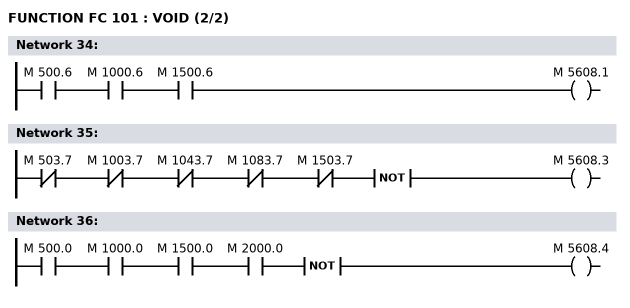

      A     M    500.6;
      A     M   1000.6;
      A     M   1500.6;
      =     M   5608.1;
NETWORK
TITLE =

      AN    M    503.7;
      AN    M   1003.7;
      AN    M   1043.7;
      AN    M   1083.7;
      AN    M   1503.7;
      NOT   ;
      =     M   5608.3;
NETWORK
TITLE =

      A     M    500.0;
      A     M   1000.0;
      A     M   1500.0;
      A     M   2000.0;
      NOT   ;
      =     M   5608.4;
NETWORK
TITLE =

      AN    OV;
      =     L      0.0;
      A     L      0.0;
      JNB   _001;
      L     ID  1302;
      T     MD  5610;
_001: NOP   0;
      A     L      0.0;
      JNB   _002;
      L     ID  1306;
      T     MD  5614;
_002: NOP   0;
      A     L      0.0;
      JNB   _003;
      L     ID  1310;
      T     MW  5618;
_003: NOP   0;
NETWORK
TITLE =

      AN    OV;
      =     L      0.0;
      A     L      0.0;
      A     I   1301.4;
      L     S5T#2S;
      SD    T     90;
      A     L      0.0;
      AN    I   1301.4;
      L     S5T#2S;
      SD    T     91;
NETWORK
TITLE =
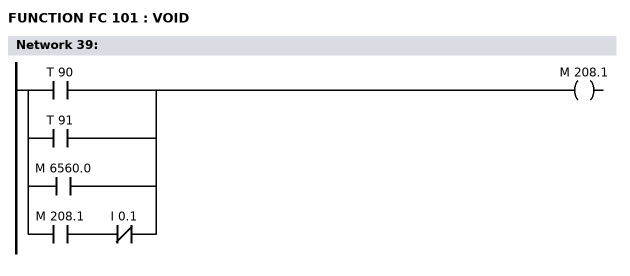

      O     T     90;
      O     T     91;
      O     M   6560.0;
      O     ;
      A     M    208.1;
      AN    I      0.1;
      =     M    208.1;
END_FUNCTION

FUNCTION_BLOCK FB 108
TITLE =
VERSION : 0.1

BEGIN
NETWORK
TITLE =PROFINET ERROR(1~10)
//
//
      A     M      3.3;
      =     L      0.0;
      A     L      0.0;
      A(    ;
      O     DB327.DBX 1025.3;
      O     ;
      A     M   7000.0;
      AN    I      0.1;
      AN    I    113.3;
      AN    I    317.3;
      AN    I    205.3;
      )     ;
      =     L      0.1;
      A     L      0.1;
      A     T    700;
      =     M   7000.0;
      A     L      0.1;
      BLD   102;
      L     S5T#0MS;
      SD    T    700;
      A     L      0.0;
      A(    ;
      O     DB327.DBX 1027.3;
      O     ;
      A     M   7000.1;
      AN    I      0.1;
      AN    I    113.3;
      AN    I    317.3;
      AN    I    205.3;
      )     ;
      =     L      0.1;
      A     L      0.1;
      A     T    701;
      =     M   7000.1;
      A     L      0.1;
      BLD   102;
      L     S5T#0MS;
      SD    T    701;
      A     L      0.0;
      A(    ;
      O     DB327.DBX 1029.3;
      O     ;
      A     M   7000.2;
      AN    I      0.1;
      AN    I    113.3;
      AN    I    317.3;
      AN    I    205.3;
      )     ;
      =     L      0.1;
      A     L      0.1;
      A     T    702;
      =     M   7000.2;
      A     L      0.1;
      BLD   102;
      L     S5T#0MS;
      SD    T    702;
      A     L      0.0;
      A(    ;
      O     DB327.DBX 1031.3;
      O     ;
      A     M   7000.3;
      AN    I      0.1;
      AN    I    113.3;
      AN    I    317.3;
      AN    I    205.3;
      )     ;
      =     L      0.1;
      A     L      0.1;
      A     T    703;
      =     M   7000.3;
      A     L      0.1;
      BLD   102;
      L     S5T#0MS;
      SD    T    703;
      A     L      0.0;
      A(    ;
      O     DB327.DBX 1033.3;
      O     ;
      A     M   7000.4;
      AN    I      0.1;
      AN    I    113.3;
      AN    I    317.3;
      AN    I    205.3;
      )     ;
      =     L      0.1;
      A     L      0.1;
      A     T    704;
      =     M   7000.4;
      A     L      0.1;
      BLD   102;
      L     S5T#0MS;
      SD    T    704;
      A     L      0.0;
      A(    ;
      O     DB327.DBX 1035.3;
      O     ;
      A     M   7000.5;
      AN    I      0.1;
      AN    I    113.3;
      AN    I    317.3;
      AN    I    205.3;
      )     ;
      =     L      0.1;
      A     L      0.1;
      A     T    705;
      =     M   7000.5;
      A     L      0.1;
      BLD   102;
      L     S5T#0MS;
      SD    T    705;
      A     L      0.0;
      A(    ;
      O     DB327.DBX 1037.3;
      O     ;
      A     M   7000.6;
      AN    I      0.1;
      AN    I    113.3;
      AN    I    317.3;
      AN    I    205.3;
      )     ;
      =     L      0.1;
      A     L      0.1;
      A     T    706;
      =     M   7000.6;
      A     L      0.1;
      BLD   102;
      L     S5T#0MS;
      SD    T    706;
      A     L      0.0;
      A(    ;
      O     DB327.DBX 1039.3;
      O     ;
      A     M   7000.7;
      AN    I      0.1;
      AN    I    113.3;
      AN    I    317.3;
      AN    I    205.3;
      )     ;
      =     L      0.1;
      A     L      0.1;
      A     T    707;
      =     M   7000.7;
      A     L      0.1;
      BLD   102;
      L     S5T#0MS;
      SD    T    707;
      A     L      0.0;
      A(    ;
      O     DB327.DBX 1041.3;
      O     ;
      A     M   7001.0;
      AN    I      0.1;
      AN    I    113.3;
      AN    I    317.3;
      AN    I    205.3;
      )     ;
      =     L      0.1;
      A     L      0.1;
      A     T    708;
      =     M   7001.0;
      A     L      0.1;
      BLD   102;
      L     S5T#0MS;
      SD    T    708;
      A     L      0.0;
      A(    ;
      O     DB327.DBX 1043.3;
      O     ;
      A     M   7001.1;
      AN    I      0.1;
      AN    I    113.3;
      AN    I    317.3;
      AN    I    205.3;
      )     ;
      =     L      0.1;
      A     L      0.1;
      A     T    709;
      =     M   7001.1;
      A     L      0.1;
      BLD   102;
      L     S5T#0MS;
      SD    T    709;
NETWORK
TITLE =PROFINET ERROR(11~20)
//
//
      A     M      3.3;
      =     L      0.0;
      A     L      0.0;
      A(    ;
      O     DB327.DBX 1045.3;
      O     ;
      A     M   7001.2;
      AN    I      0.1;
      AN    I    113.3;
      AN    I    317.3;
      AN    I    205.3;
      )     ;
      =     L      0.1;
      A     L      0.1;
      A     T    710;
      =     M   7001.2;
      A     L      0.1;
      BLD   102;
      L     S5T#0MS;
      SD    T    710;
      A     L      0.0;
      A(    ;
      O     DB327.DBX 1047.3;
      O     ;
      A     M   7001.3;
      AN    I      0.1;
      AN    I    113.3;
      AN    I    317.3;
      AN    I    205.3;
      )     ;
      =     L      0.1;
      A     L      0.1;
      A     T    711;
      =     M   7001.3;
      A     L      0.1;
      BLD   102;
      L     S5T#0MS;
      SD    T    711;
      A     L      0.0;
      A(    ;
      O     DB327.DBX 1049.3;
      O     ;
      A     M   7001.4;
      AN    I      0.1;
      AN    I    113.3;
      AN    I    317.3;
      AN    I    205.3;
      )     ;
      =     L      0.1;
      A     L      0.1;
      A     T    712;
      =     M   7001.4;
      A     L      0.1;
      BLD   102;
      L     S5T#0MS;
      SD    T    712;
      A     L      0.0;
      A(    ;
      O     DB327.DBX 1051.3;
      O     ;
      A     M   7001.5;
      AN    I      0.1;
      AN    I    113.3;
      AN    I    317.3;
      AN    I    205.3;
      )     ;
      =     L      0.1;
      A     L      0.1;
      A     T    713;
      =     M   7001.5;
      A     L      0.1;
      BLD   102;
      L     S5T#0MS;
      SD    T    713;
      A     L      0.0;
      A(    ;
      O     DB327.DBX 1053.3;
      O     ;
      A     M   7001.6;
      AN    I      0.1;
      AN    I    113.3;
      AN    I    317.3;
      AN    I    205.3;
      )     ;
      =     L      0.1;
      A     L      0.1;
      A     T    714;
      =     M   7001.6;
      A     L      0.1;
      BLD   102;
      L     S5T#0MS;
      SD    T    714;
      A     L      0.0;
      A(    ;
      O     DB327.DBX 1055.3;
      O     ;
      A     M   7001.7;
      AN    I      0.1;
      AN    I    113.3;
      AN    I    317.3;
      AN    I    205.3;
      )     ;
      =     L      0.1;
      A     L      0.1;
      A     T    715;
      =     M   7001.7;
      A     L      0.1;
      BLD   102;
      L     S5T#0MS;
      SD    T    715;
      A     L      0.0;
      A(    ;
      O     DB327.DBX 1057.3;
      O     ;
      A     M   7002.0;
      AN    I      0.1;
      AN    I    113.3;
      AN    I    317.3;
      AN    I    205.3;
      )     ;
      =     L      0.1;
      A     L      0.1;
      A     T    716;
      =     M   7002.0;
      A     L      0.1;
      BLD   102;
      L     S5T#0MS;
      SD    T    716;
      A     L      0.0;
      A(    ;
      O     DB327.DBX 1059.3;
      O     ;
      A     M   7002.1;
      AN    I      0.1;
      AN    I    113.3;
      AN    I    317.3;
      AN    I    205.3;
      )     ;
      =     L      0.1;
      A     L      0.1;
      A     T    717;
      =     M   7002.1;
      A     L      0.1;
      BLD   102;
      L     S5T#0MS;
      SD    T    717;
      A     L      0.0;
      A(    ;
      O     DB327.DBX 1061.3;
      O     ;
      A     M   7002.2;
      AN    I      0.1;
      AN    I    113.3;
      AN    I    317.3;
      AN    I    205.3;
      )     ;
      =     L      0.1;
      A     L      0.1;
      A     T    718;
      =     M   7002.2;
      A     L      0.1;
      BLD   102;
      L     S5T#0MS;
      SD    T    718;
      A     L      0.0;
      A(    ;
      O     DB327.DBX 1063.3;
      O     ;
      A     M   7002.3;
      AN    I      0.1;
      AN    I    113.3;
      AN    I    317.3;
      AN    I    205.3;
      )     ;
      =     L      0.1;
      A     L      0.1;
      A     T    719;
      =     M   7002.3;
      A     L      0.1;
      BLD   102;
      L     S5T#0MS;
      SD    T    719;
NETWORK
TITLE =PROFINET ERROR(21~30)
//
//
      A     M      3.3;
      =     L      0.0;
      A     L      0.0;
      A(    ;
      O     DB327.DBX 1065.3;
      O     ;
      A     M   7002.4;
      AN    I      0.1;
      AN    I    113.3;
      AN    I    317.3;
      AN    I    205.3;
      )     ;
      =     L      0.1;
      A     L      0.1;
      A     T    720;
      =     M   7002.4;
      A     L      0.1;
      BLD   102;
      L     S5T#0MS;
      SD    T    720;
      A     L      0.0;
      A(    ;
      O     DB327.DBX 1067.3;
      O     ;
      A     M   7002.5;
      AN    I      0.1;
      AN    I    113.3;
      AN    I    317.3;
      AN    I    205.3;
      )     ;
      =     L      0.1;
      A     L      0.1;
      A     T    721;
      =     M   7002.5;
      A     L      0.1;
      BLD   102;
      L     S5T#0MS;
      SD    T    721;
      A     L      0.0;
      A(    ;
      O     DB327.DBX 1069.3;
      O     ;
      A     M   7002.6;
      AN    I      0.1;
      AN    I    113.3;
      AN    I    317.3;
      AN    I    205.3;
      )     ;
      =     L      0.1;
      A     L      0.1;
      A     T    722;
      =     M   7002.6;
      A     L      0.1;
      BLD   102;
      L     S5T#0MS;
      SD    T    722;
      A     L      0.0;
      A(    ;
      O     DB327.DBX 1071.3;
      O     ;
      A     M   7002.7;
      AN    I      0.1;
      AN    I    113.3;
      AN    I    317.3;
      AN    I    205.3;
      )     ;
      =     L      0.1;
      A     L      0.1;
      A     T    723;
      =     M   7002.7;
      A     L      0.1;
      BLD   102;
      L     S5T#0MS;
      SD    T    723;
      A     L      0.0;
      A(    ;
      O     DB327.DBX 1073.3;
      O     ;
      A     M   7003.0;
      AN    I      0.1;
      AN    I    113.3;
      AN    I    317.3;
      AN    I    205.3;
      )     ;
      =     L      0.1;
      A     L      0.1;
      A     T    724;
      =     M   7003.0;
      A     L      0.1;
      BLD   102;
      L     S5T#0MS;
      SD    T    724;
      A     L      0.0;
      A(    ;
      O     DB327.DBX 1075.3;
      O     ;
      A     M   7003.1;
      AN    I      0.1;
      AN    I    113.3;
      AN    I    317.3;
      AN    I    205.3;
      )     ;
      =     L      0.1;
      A     L      0.1;
      A     T    725;
      =     M   7003.1;
      A     L      0.1;
      BLD   102;
      L     S5T#0MS;
      SD    T    725;
      A     L      0.0;
      A(    ;
      O     DB327.DBX 1077.3;
      O     ;
      A     M   7003.2;
      AN    I      0.1;
      AN    I    113.3;
      AN    I    317.3;
      AN    I    205.3;
      )     ;
      =     L      0.1;
      A     L      0.1;
      A     T    726;
      AN    M      3.3;
      =     M   7003.2;
      A     L      0.1;
      BLD   102;
      L     S5T#0MS;
      SD    T    726;
      A     L      0.0;
      A(    ;
      O     DB327.DBX 1079.3;
      O     ;
      A     M   7003.3;
      AN    I      0.1;
      AN    I    113.3;
      AN    I    317.3;
      AN    I    205.3;
      )     ;
      =     L      0.1;
      A     L      0.1;
      A     T    727;
      AN    M      3.3;
      =     M   7003.3;
      A     L      0.1;
      BLD   102;
      L     S5T#0MS;
      SD    T    727;
      A     L      0.0;
      A(    ;
      O     DB327.DBX 1081.3;
      O     ;
      A     M   7003.4;
      AN    I      0.1;
      AN    I    113.3;
      AN    I    317.3;
      AN    I    205.3;
      )     ;
      =     L      0.1;
      A     L      0.1;
      A     T    728;
      AN    M      3.3;
      =     M   7003.4;
      A     L      0.1;
      BLD   102;
      L     S5T#0MS;
      SD    T    728;
      A     L      0.0;
      A(    ;
      O     DB327.DBX 1083.3;
      O     ;
      A     M   7003.5;
      AN    I      0.1;
      AN    I    113.3;
      AN    I    317.3;
      AN    I    205.3;
      )     ;
      =     L      0.1;
      A     L      0.1;
      A     T    729;
      AN    M      3.3;
      =     M   7003.5;
      A     L      0.1;
      BLD   102;
      L     S5T#0MS;
      SD    T    729;
NETWORK
TITLE =PROFINET ERROR(31~40)
//
//
      A     M      3.3;
      =     L      0.0;
      A     L      0.0;
      A(    ;
      O     DB327.DBX 1085.3;
      O     ;
      A     M   7003.6;
      AN    I      0.1;
      AN    I    113.3;
      AN    I    317.3;
      AN    I    205.3;
      )     ;
      =     L      0.1;
      A     L      0.1;
      A     T    730;
      AN    M      3.3;
      =     M   7003.6;
      A     L      0.1;
      BLD   102;
      L     S5T#0MS;
      SD    T    730;
      A     L      0.0;
      A(    ;
      O     DB327.DBX 1087.3;
      O     ;
      A     M   7003.7;
      AN    I      0.1;
      AN    I    113.3;
      AN    I    317.3;
      AN    I    205.3;
      )     ;
      =     L      0.1;
      A     L      0.1;
      A     T    731;
      AN    M      3.3;
      =     M   7003.7;
      A     L      0.1;
      BLD   102;
      L     S5T#0MS;
      SD    T    731;
      A     L      0.0;
      A(    ;
      O     DB327.DBX 1089.3;
      O     ;
      A     M   7004.0;
      AN    I      0.1;
      AN    I    113.3;
      AN    I    317.3;
      AN    I    205.3;
      )     ;
      =     L      0.1;
      A     L      0.1;
      A     T    732;
      AN    M      3.3;
      =     M   7004.0;
      A     L      0.1;
      BLD   102;
      L     S5T#0MS;
      SD    T    732;
      A     L      0.0;
      A(    ;
      O     DB327.DBX 1091.3;
      O     ;
      A     M   7004.1;
      AN    I      0.1;
      AN    I    113.3;
      AN    I    317.3;
      AN    I    205.3;
      )     ;
      =     L      0.1;
      A     L      0.1;
      A     T    733;
      AN    M      3.3;
      =     M   7004.1;
      A     L      0.1;
      BLD   102;
      L     S5T#0MS;
      SD    T    733;
      A     L      0.0;
      A(    ;
      O     DB327.DBX 1093.3;
      O     ;
      A     M   7004.2;
      AN    I      0.1;
      AN    I    113.3;
      AN    I    317.3;
      AN    I    205.3;
      )     ;
      =     L      0.1;
      A     L      0.1;
      A     T    734;
      AN    M      3.3;
      =     M   7004.2;
      A     L      0.1;
      BLD   102;
      L     S5T#0MS;
      SD    T    734;
      A     L      0.0;
      A(    ;
      O     DB327.DBX 1095.3;
      O     ;
      A     M   7004.3;
      AN    I      0.1;
      AN    I    113.3;
      AN    I    317.3;
      AN    I    205.3;
      )     ;
      =     L      0.1;
      A     L      0.1;
      A     T    735;
      AN    M      3.3;
      =     M   7004.3;
      A     L      0.1;
      BLD   102;
      L     S5T#0MS;
      SD    T    735;
      A     L      0.0;
      A(    ;
      O     DB327.DBX 1097.3;
      O     ;
      A     M   7004.4;
      AN    I      0.1;
      AN    I    113.3;
      AN    I    317.3;
      AN    I    205.3;
      )     ;
      =     L      0.1;
      A     L      0.1;
      A     T    736;
      AN    M      3.3;
      =     M   7004.4;
      A     L      0.1;
      BLD   102;
      L     S5T#0MS;
      SD    T    736;
      A     L      0.0;
      A(    ;
      O     DB327.DBX 1099.3;
      O     ;
      A     M   7004.5;
      AN    I      0.1;
      AN    I    113.3;
      AN    I    317.3;
      AN    I    205.3;
      )     ;
      =     L      0.1;
      A     L      0.1;
      A     T    737;
      AN    M      3.3;
      =     M   7004.5;
      A     L      0.1;
      BLD   102;
      L     S5T#0MS;
      SD    T    737;
      A     L      0.0;
      A(    ;
      O     DB327.DBX 1101.3;
      O     ;
      A     M   7004.6;
      AN    I      0.1;
      AN    I    113.3;
      AN    I    317.3;
      AN    I    205.3;
      )     ;
      =     L      0.1;
      A     L      0.1;
      A     T    738;
      AN    M      3.3;
      =     M   7004.6;
      A     L      0.1;
      BLD   102;
      L     S5T#0MS;
      SD    T    738;
      A     L      0.0;
      A(    ;
      O     DB327.DBX 1103.3;
      O     ;
      A     M   7004.7;
      AN    I      0.1;
      AN    I    113.3;
      AN    I    317.3;
      AN    I    205.3;
      )     ;
      =     L      0.1;
      A     L      0.1;
      A     T    739;
      AN    M      3.3;
      =     M   7004.7;
      A     L      0.1;
      BLD   102;
      L     S5T#0MS;
      SD    T    739;
NETWORK
TITLE =PROFINET ERROR(150~159)

      A     M      3.3;
      =     L      0.0;
      A     L      0.0;
      A(    ;
      O     DB327.DBX 1323.3;
      O     ;
      A     M   7018.5;
      AN    I      0.1;
      AN    I    113.3;
      AN    I    317.3;
      AN    I    205.3;
      )     ;
      =     L      0.1;
      A     L      0.1;
      A     T    849;
      =     M   7018.5;
      A     L      0.1;
      BLD   102;
      L     S5T#0MS;
      SD    T    849;
      A     L      0.0;
      A(    ;
      O     DB327.DBX 1325.3;
      O     ;
      A     M   7018.6;
      AN    I      0.1;
      AN    I    113.3;
      AN    I    317.3;
      AN    I    205.3;
      )     ;
      =     L      0.1;
      A     L      0.1;
      A     T    850;
      =     M   7018.6;
      A     L      0.1;
      BLD   102;
      L     S5T#0MS;
      SD    T    850;
      A     L      0.0;
      A(    ;
      O     DB327.DBX 1327.3;
      O     ;
      A     M   7018.7;
      AN    I      0.1;
      AN    I    113.3;
      AN    I    317.3;
      AN    I    205.3;
      )     ;
      =     L      0.1;
      A     L      0.1;
      A     T    851;
      =     M   7018.7;
      A     L      0.1;
      BLD   102;
      L     S5T#0MS;
      SD    T    851;
      A     L      0.0;
      A(    ;
      O     DB327.DBX 1329.3;
      O     ;
      A     M   7019.0;
      AN    I      0.1;
      AN    I    113.3;
      AN    I    317.3;
      AN    I    205.3;
      )     ;
      =     L      0.1;
      A     L      0.1;
      A     T    852;
      =     M   7019.0;
      A     L      0.1;
      BLD   102;
      L     S5T#0MS;
      SD    T    852;
      A     L      0.0;
      A(    ;
      O     DB327.DBX 1331.3;
      O     ;
      A     M   7019.1;
      AN    I      0.1;
      AN    I    113.3;
      AN    I    317.3;
      AN    I    205.3;
      )     ;
      =     L      0.1;
      A     L      0.1;
      A     T    853;
      =     M   7019.1;
      A     L      0.1;
      BLD   102;
      L     S5T#0MS;
      SD    T    853;
      A     L      0.0;
      A(    ;
      O     DB327.DBX 1333.3;
      O     ;
      A     M   7019.2;
      AN    I      0.1;
      AN    I    113.3;
      AN    I    317.3;
      AN    I    205.3;
      )     ;
      =     L      0.1;
      A     L      0.1;
      A     T    854;
      =     M   7019.2;
      A     L      0.1;
      BLD   102;
      L     S5T#0MS;
      SD    T    854;
      A     L      0.0;
      A(    ;
      O     DB327.DBX 1335.3;
      O     ;
      A     M   7019.3;
      AN    I      0.1;
      AN    I    113.3;
      AN    I    317.3;
      AN    I    205.3;
      )     ;
      =     L      0.1;
      A     L      0.1;
      A     T    855;
      AN    M      3.3;
      =     M   7019.3;
      A     L      0.1;
      BLD   102;
      L     S5T#0MS;
      SD    T    855;
      A     L      0.0;
      A(    ;
      O     DB327.DBX 1337.3;
      O     ;
      A     M   7019.4;
      AN    I      0.1;
      AN    I    113.3;
      AN    I    317.3;
      AN    I    205.3;
      )     ;
      =     L      0.1;
      A     L      0.1;
      A     T    856;
      AN    M      3.3;
      =     M   7019.4;
      A     L      0.1;
      BLD   102;
      L     S5T#0MS;
      SD    T    856;
      A     L      0.0;
      A(    ;
      O     DB327.DBX 1339.3;
      O     ;
      A     M   7019.5;
      AN    I      0.1;
      AN    I    113.3;
      AN    I    317.3;
      AN    I    205.3;
      )     ;
      =     L      0.1;
      A     L      0.1;
      A     T    857;
      AN    M      3.3;
      =     M   7019.5;
      A     L      0.1;
      BLD   102;
      L     S5T#0MS;
      SD    T    857;
      A     L      0.0;
      A(    ;
      O     DB327.DBX 1341.3;
      O     ;
      A     M   7019.6;
      AN    I      0.1;
      AN    I    113.3;
      AN    I    317.3;
      AN    I    205.3;
      )     ;
      =     L      0.1;
      A     L      0.1;
      A     T    858;
      AN    M      3.3;
      =     M   7019.6;
      A     L      0.1;
      BLD   102;
      L     S5T#0MS;
      SD    T    858;
NETWORK
TITLE =CP TRIP(20~29)
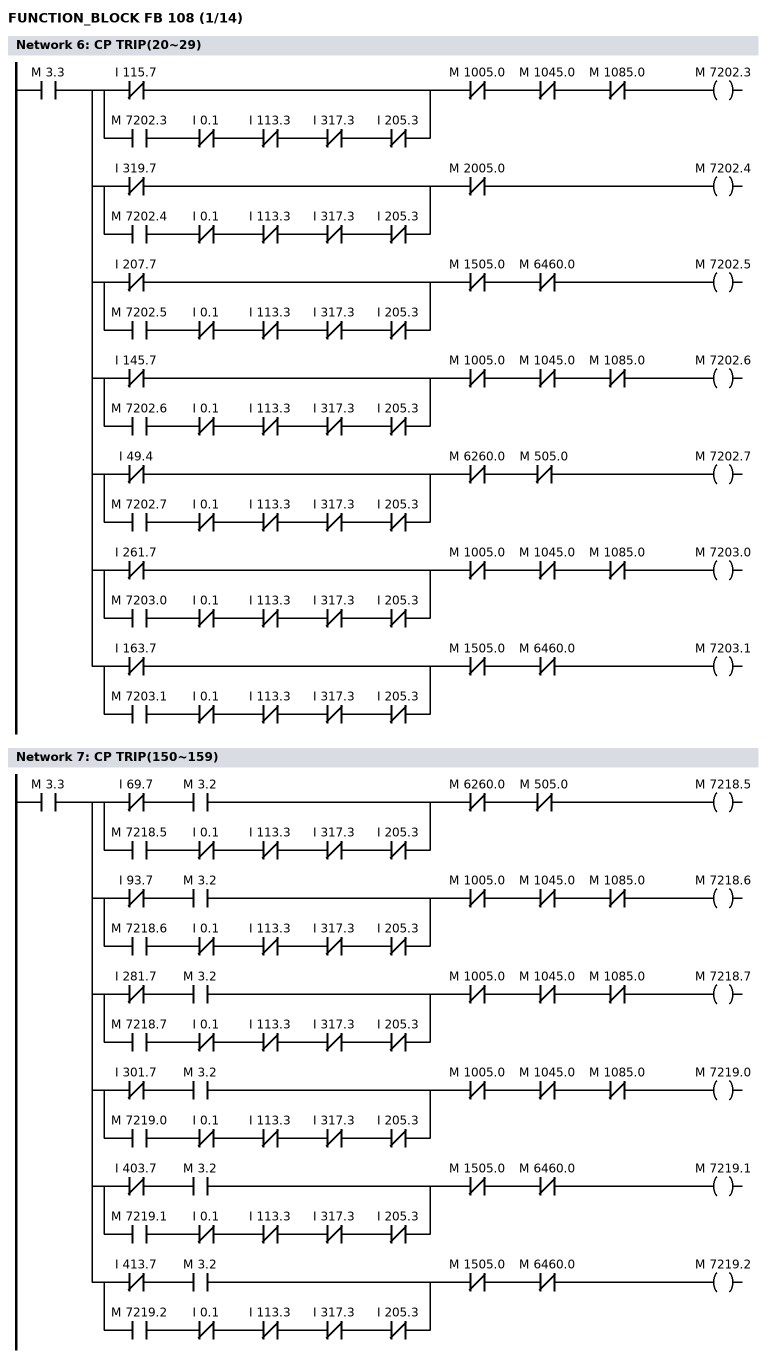

      A     M      3.3;
      =     L      0.0;
      A     L      0.0;
      A(    ;
      ON    I    115.7;
      O     ;
      A     M   7202.3;
      AN    I      0.1;
      AN    I    113.3;
      AN    I    317.3;
      AN    I    205.3;
      )     ;
      AN    M   1005.0;
      AN    M   1045.0;
      AN    M   1085.0;
      =     M   7202.3;
      A     L      0.0;
      A(    ;
      ON    I    319.7;
      O     ;
      A     M   7202.4;
      AN    I      0.1;
      AN    I    113.3;
      AN    I    317.3;
      AN    I    205.3;
      )     ;
      AN    M   2005.0;
      =     M   7202.4;
      A     L      0.0;
      A(    ;
      ON    I    207.7;
      O     ;
      A     M   7202.5;
      AN    I      0.1;
      AN    I    113.3;
      AN    I    317.3;
      AN    I    205.3;
      )     ;
      AN    M   1505.0;
      AN    M   6460.0;
      =     M   7202.5;
      A     L      0.0;
      A(    ;
      ON    I    145.7;
      O     ;
      A     M   7202.6;
      AN    I      0.1;
      AN    I    113.3;
      AN    I    317.3;
      AN    I    205.3;
      )     ;
      AN    M   1005.0;
      AN    M   1045.0;
      AN    M   1085.0;
      =     M   7202.6;
      A     L      0.0;
      A(    ;
      ON    I     49.4;
      O     ;
      A     M   7202.7;
      AN    I      0.1;
      AN    I    113.3;
      AN    I    317.3;
      AN    I    205.3;
      )     ;
      AN    M   6260.0;
      AN    M    505.0;
      =     M   7202.7;
      A     L      0.0;
      A(    ;
      ON    I    261.7;
      O     ;
      A     M   7203.0;
      AN    I      0.1;
      AN    I    113.3;
      AN    I    317.3;
      AN    I    205.3;
      )     ;
      AN    M   1005.0;
      AN    M   1045.0;
      AN    M   1085.0;
      =     M   7203.0;
      A     L      0.0;
      A(    ;
      ON    I    163.7;
      O     ;
      A     M   7203.1;
      AN    I      0.1;
      AN    I    113.3;
      AN    I    317.3;
      AN    I    205.3;
      )     ;
      AN    M   1505.0;
      AN    M   6460.0;
      =     M   7203.1;
NETWORK
TITLE =CP TRIP(150~159)

      A     M      3.3;
      =     L      0.0;
      A     L      0.0;
      A(    ;
      AN    I     69.7;
      A     M      3.2;
      O     ;
      A     M   7218.5;
      AN    I      0.1;
      AN    I    113.3;
      AN    I    317.3;
      AN    I    205.3;
      )     ;
      AN    M   6260.0;
      AN    M    505.0;
      =     M   7218.5;
      A     L      0.0;
      A(    ;
      AN    I     93.7;
      A     M      3.2;
      O     ;
      A     M   7218.6;
      AN    I      0.1;
      AN    I    113.3;
      AN    I    317.3;
      AN    I    205.3;
      )     ;
      AN    M   1005.0;
      AN    M   1045.0;
      AN    M   1085.0;
      =     M   7218.6;
      A     L      0.0;
      A(    ;
      AN    I    281.7;
      A     M      3.2;
      O     ;
      A     M   7218.7;
      AN    I      0.1;
      AN    I    113.3;
      AN    I    317.3;
      AN    I    205.3;
      )     ;
      AN    M   1005.0;
      AN    M   1045.0;
      AN    M   1085.0;
      =     M   7218.7;
      A     L      0.0;
      A(    ;
      AN    I    301.7;
      A     M      3.2;
      O     ;
      A     M   7219.0;
      AN    I      0.1;
      AN    I    113.3;
      AN    I    317.3;
      AN    I    205.3;
      )     ;
      AN    M   1005.0;
      AN    M   1045.0;
      AN    M   1085.0;
      =     M   7219.0;
      A     L      0.0;
      A(    ;
      AN    I    403.7;
      A     M      3.2;
      O     ;
      A     M   7219.1;
      AN    I      0.1;
      AN    I    113.3;
      AN    I    317.3;
      AN    I    205.3;
      )     ;
      AN    M   1505.0;
      AN    M   6460.0;
      =     M   7219.1;
      A     L      0.0;
      A(    ;
      AN    I    413.7;
      A     M      3.2;
      O     ;
      A     M   7219.2;
      AN    I      0.1;
      AN    I    113.3;
      AN    I    317.3;
      AN    I    205.3;
      )     ;
      AN    M   1505.0;
      AN    M   6460.0;
      =     M   7219.2;
NETWORK
TITLE =통신확인 비트(M4301.0) 1초 플리커
//
//
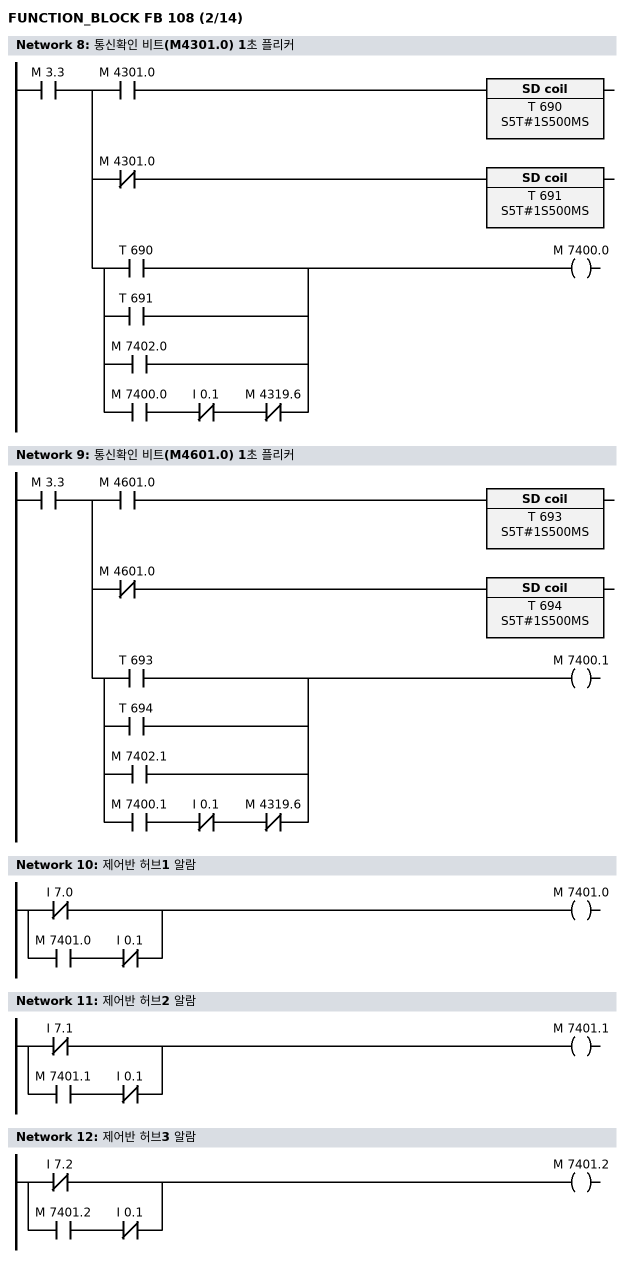
      A     M      3.3;
      =     L      0.0;
      A     L      0.0;
      A     M   4301.0;
      L     S5T#1S500MS;
      SD    T    690;
      A     L      0.0;
      AN    M   4301.0;
      L     S5T#1S500MS;
      SD    T    691;
      A     L      0.0;
      A(    ;
      O     T    690;
      O     T    691;
      O     M   7402.0;
      O     ;
      A     M   7400.0;
      AN    I      0.1;
      AN    M   4319.6;
      )     ;
      =     M   7400.0;
NETWORK
TITLE =통신확인 비트(M4601.0) 1초 플리커
//
//
//
      A     M      3.3;
      =     L      0.0;
      A     L      0.0;
      A     M   4601.0;
      L     S5T#1S500MS;
      SD    T    693;
      A     L      0.0;
      AN    M   4601.0;
      L     S5T#1S500MS;
      SD    T    694;
      A     L      0.0;
      A(    ;
      O     T    693;
      O     T    694;
      O     M   7402.1;
      O     ;
      A     M   7400.1;
      AN    I      0.1;
      AN    M   4319.6;
      )     ;
      =     M   7400.1;
NETWORK
TITLE =제어반 허브1 알람

      ON    I      7.0;
      O     ;
      A     M   7401.0;
      AN    I      0.1;
      =     M   7401.0;
NETWORK
TITLE =제어반 허브2 알람

      ON    I      7.1;
      O     ;
      A     M   7401.1;
      AN    I      0.1;
      =     M   7401.1;
NETWORK
TITLE =제어반 허브3 알람

      ON    I      7.2;
      O     ;
      A     M   7401.2;
      AN    I      0.1;
      =     M   7401.2;
NETWORK
TITLE =제어반 POWER SUPPLY1 알람
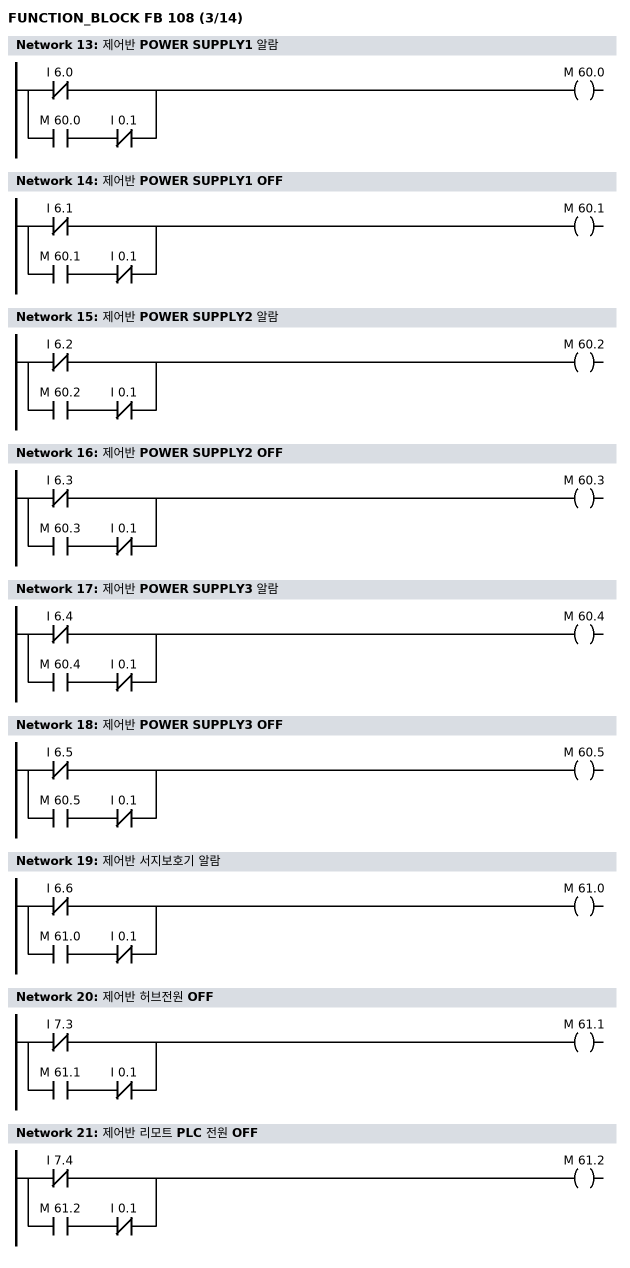

      ON    I      6.0;
      O     ;
      A     M     60.0;
      AN    I      0.1;
      =     M     60.0;
NETWORK
TITLE =제어반 POWER SUPPLY1 OFF

      ON    I      6.1;
      O     ;
      A     M     60.1;
      AN    I      0.1;
      =     M     60.1;
NETWORK
TITLE =제어반 POWER SUPPLY2 알람
//
//
      ON    I      6.2;
      O     ;
      A     M     60.2;
      AN    I      0.1;
      =     M     60.2;
NETWORK
TITLE =제어반 POWER SUPPLY2 OFF

      ON    I      6.3;
      O     ;
      A     M     60.3;
      AN    I      0.1;
      =     M     60.3;
NETWORK
TITLE =제어반 POWER SUPPLY3 알람
//
//
      ON    I      6.4;
      O     ;
      A     M     60.4;
      AN    I      0.1;
      =     M     60.4;
NETWORK
TITLE =제어반 POWER SUPPLY3 OFF

      ON    I      6.5;
      O     ;
      A     M     60.5;
      AN    I      0.1;
      =     M     60.5;
NETWORK
TITLE =제어반 서지보호기 알람

      ON    I      6.6;
      O     ;
      A     M     61.0;
      AN    I      0.1;
      =     M     61.0;
NETWORK
TITLE =제어반 허브전원 OFF

      ON    I      7.3;
      O     ;
      A     M     61.1;
      AN    I      0.1;
      =     M     61.1;
NETWORK
TITLE =제어반 리모트 PLC 전원 OFF

      ON    I      7.4;
      O     ;
      A     M     61.2;
      AN    I      0.1;
      =     M     61.2;
NETWORK
TITLE =제어반내 I/O 전원 OFF
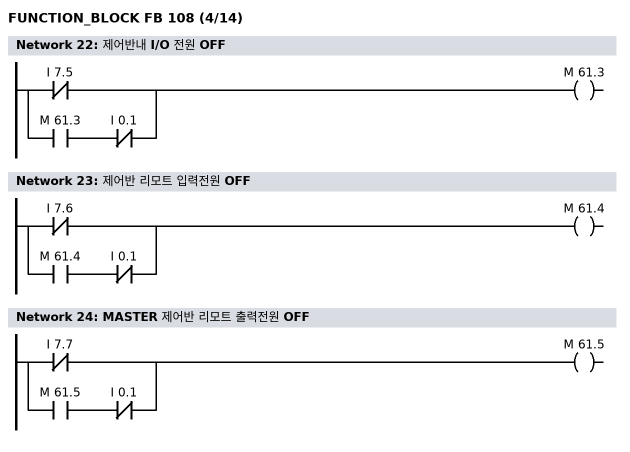

      ON    I      7.5;
      O     ;
      A     M     61.3;
      AN    I      0.1;
      =     M     61.3;
NETWORK
TITLE =제어반 리모트 입력전원 OFF

      ON    I      7.6;
      O     ;
      A     M     61.4;
      AN    I      0.1;
      =     M     61.4;
NETWORK
TITLE =MASTER 제어반 리모트 출력전원 OFF

      ON    I      7.7;
      O     ;
      A     M     61.5;
      AN    I      0.1;
      =     M     61.5;
NETWORK
TITLE =PROFINET ALARM-모듈이상이나 통신케이블단선(1~10)
//
//
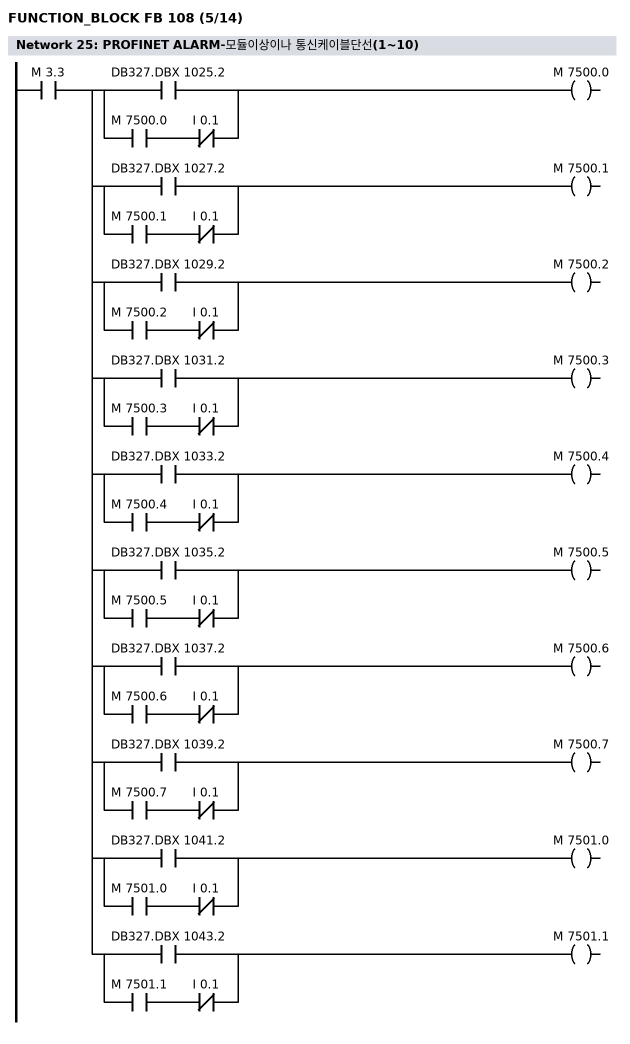
      A     M      3.3;
      =     L      0.0;
      A     L      0.0;
      A(    ;
      O     DB327.DBX 1025.2;
      O     ;
      A     M   7500.0;
      AN    I      0.1;
      )     ;
      =     M   7500.0;
      A     L      0.0;
      A(    ;
      O     DB327.DBX 1027.2;
      O     ;
      A     M   7500.1;
      AN    I      0.1;
      )     ;
      =     M   7500.1;
      A     L      0.0;
      A(    ;
      O     DB327.DBX 1029.2;
      O     ;
      A     M   7500.2;
      AN    I      0.1;
      )     ;
      =     M   7500.2;
      A     L      0.0;
      A(    ;
      O     DB327.DBX 1031.2;
      O     ;
      A     M   7500.3;
      AN    I      0.1;
      )     ;
      =     M   7500.3;
      A     L      0.0;
      A(    ;
      O     DB327.DBX 1033.2;
      O     ;
      A     M   7500.4;
      AN    I      0.1;
      )     ;
      =     M   7500.4;
      A     L      0.0;
      A(    ;
      O     DB327.DBX 1035.2;
      O     ;
      A     M   7500.5;
      AN    I      0.1;
      )     ;
      =     M   7500.5;
      A     L      0.0;
      A(    ;
      O     DB327.DBX 1037.2;
      O     ;
      A     M   7500.6;
      AN    I      0.1;
      )     ;
      =     M   7500.6;
      A     L      0.0;
      A(    ;
      O     DB327.DBX 1039.2;
      O     ;
      A     M   7500.7;
      AN    I      0.1;
      )     ;
      =     M   7500.7;
      A     L      0.0;
      A(    ;
      O     DB327.DBX 1041.2;
      O     ;
      A     M   7501.0;
      AN    I      0.1;
      )     ;
      =     M   7501.0;
      A     L      0.0;
      A(    ;
      O     DB327.DBX 1043.2;
      O     ;
      A     M   7501.1;
      AN    I      0.1;
      )     ;
      =     M   7501.1;
NETWORK
TITLE =PROFINET ALARM-모듈이상이나 통신케이블단선(11~20)
//
//
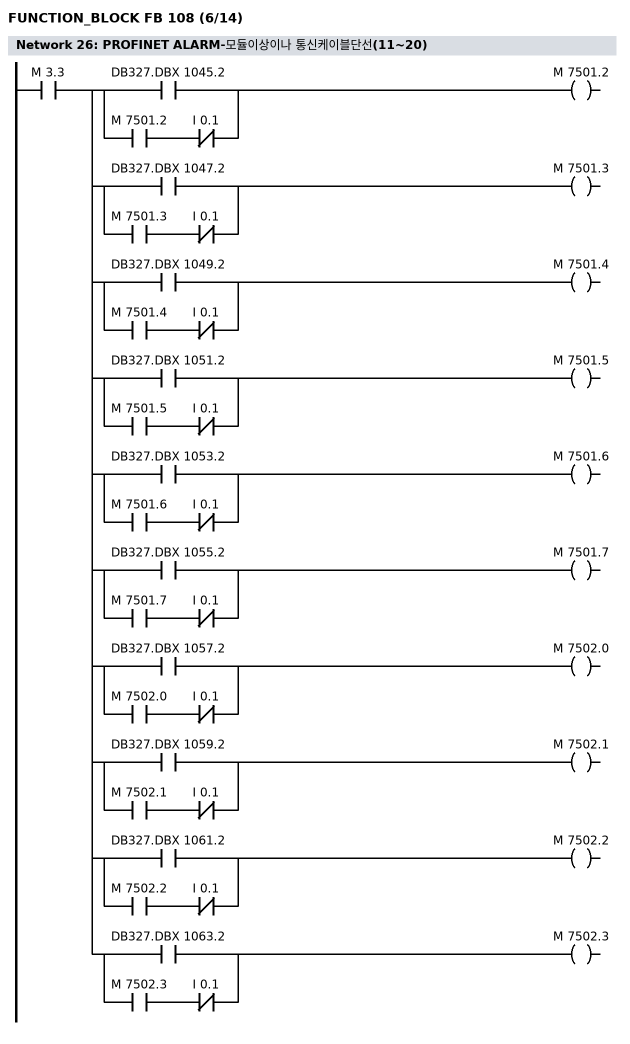
      A     M      3.3;
      =     L      0.0;
      A     L      0.0;
      A(    ;
      O     DB327.DBX 1045.2;
      O     ;
      A     M   7501.2;
      AN    I      0.1;
      )     ;
      =     M   7501.2;
      A     L      0.0;
      A(    ;
      O     DB327.DBX 1047.2;
      O     ;
      A     M   7501.3;
      AN    I      0.1;
      )     ;
      =     M   7501.3;
      A     L      0.0;
      A(    ;
      O     DB327.DBX 1049.2;
      O     ;
      A     M   7501.4;
      AN    I      0.1;
      )     ;
      =     M   7501.4;
      A     L      0.0;
      A(    ;
      O     DB327.DBX 1051.2;
      O     ;
      A     M   7501.5;
      AN    I      0.1;
      )     ;
      =     M   7501.5;
      A     L      0.0;
      A(    ;
      O     DB327.DBX 1053.2;
      O     ;
      A     M   7501.6;
      AN    I      0.1;
      )     ;
      =     M   7501.6;
      A     L      0.0;
      A(    ;
      O     DB327.DBX 1055.2;
      O     ;
      A     M   7501.7;
      AN    I      0.1;
      )     ;
      =     M   7501.7;
      A     L      0.0;
      A(    ;
      O     DB327.DBX 1057.2;
      O     ;
      A     M   7502.0;
      AN    I      0.1;
      )     ;
      =     M   7502.0;
      A     L      0.0;
      A(    ;
      O     DB327.DBX 1059.2;
      O     ;
      A     M   7502.1;
      AN    I      0.1;
      )     ;
      =     M   7502.1;
      A     L      0.0;
      A(    ;
      O     DB327.DBX 1061.2;
      O     ;
      A     M   7502.2;
      AN    I      0.1;
      )     ;
      =     M   7502.2;
      A     L      0.0;
      A(    ;
      O     DB327.DBX 1063.2;
      O     ;
      A     M   7502.3;
      AN    I      0.1;
      )     ;
      =     M   7502.3;
NETWORK
TITLE =PROFINET ALARM-모듈이상이나 통신케이블단선(21~30)
//
//
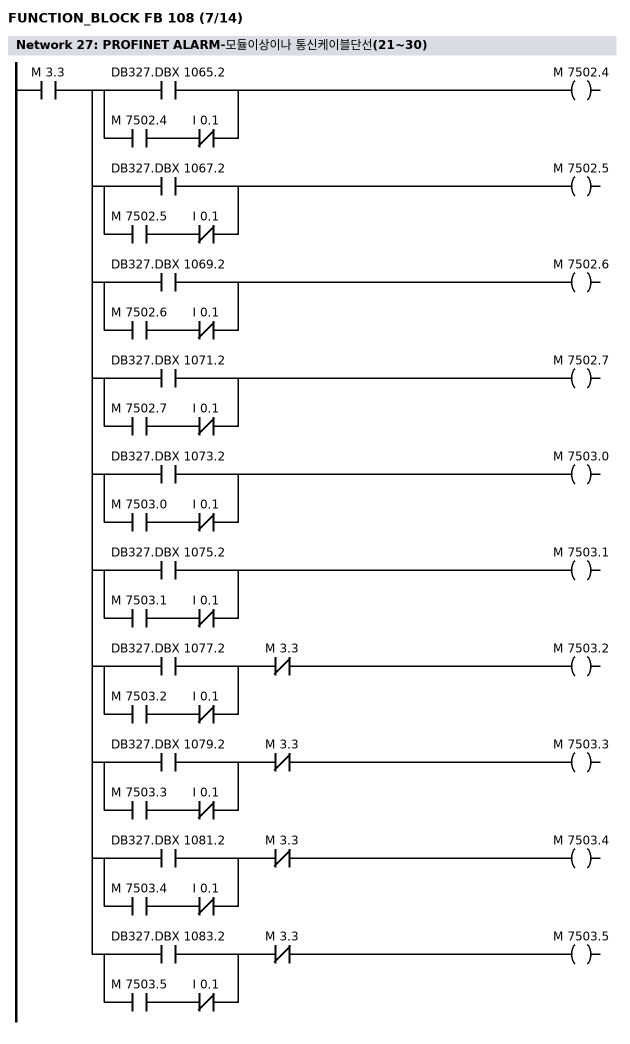
      A     M      3.3;
      =     L      0.0;
      A     L      0.0;
      A(    ;
      O     DB327.DBX 1065.2;
      O     ;
      A     M   7502.4;
      AN    I      0.1;
      )     ;
      =     M   7502.4;
      A     L      0.0;
      A(    ;
      O     DB327.DBX 1067.2;
      O     ;
      A     M   7502.5;
      AN    I      0.1;
      )     ;
      =     M   7502.5;
      A     L      0.0;
      A(    ;
      O     DB327.DBX 1069.2;
      O     ;
      A     M   7502.6;
      AN    I      0.1;
      )     ;
      =     M   7502.6;
      A     L      0.0;
      A(    ;
      O     DB327.DBX 1071.2;
      O     ;
      A     M   7502.7;
      AN    I      0.1;
      )     ;
      =     M   7502.7;
      A     L      0.0;
      A(    ;
      O     DB327.DBX 1073.2;
      O     ;
      A     M   7503.0;
      AN    I      0.1;
      )     ;
      =     M   7503.0;
      A     L      0.0;
      A(    ;
      O     DB327.DBX 1075.2;
      O     ;
      A     M   7503.1;
      AN    I      0.1;
      )     ;
      =     M   7503.1;
      A     L      0.0;
      A(    ;
      O     DB327.DBX 1077.2;
      O     ;
      A     M   7503.2;
      AN    I      0.1;
      )     ;
      AN    M      3.3;
      =     M   7503.2;
      A     L      0.0;
      A(    ;
      O     DB327.DBX 1079.2;
      O     ;
      A     M   7503.3;
      AN    I      0.1;
      )     ;
      AN    M      3.3;
      =     M   7503.3;
      A     L      0.0;
      A(    ;
      O     DB327.DBX 1081.2;
      O     ;
      A     M   7503.4;
      AN    I      0.1;
      )     ;
      AN    M      3.3;
      =     M   7503.4;
      A     L      0.0;
      A(    ;
      O     DB327.DBX 1083.2;
      O     ;
      A     M   7503.5;
      AN    I      0.1;
      )     ;
      AN    M      3.3;
      =     M   7503.5;
NETWORK
TITLE =PROFINET ALARM-모듈이상이나 통신케이블단선(31~40)
//
//
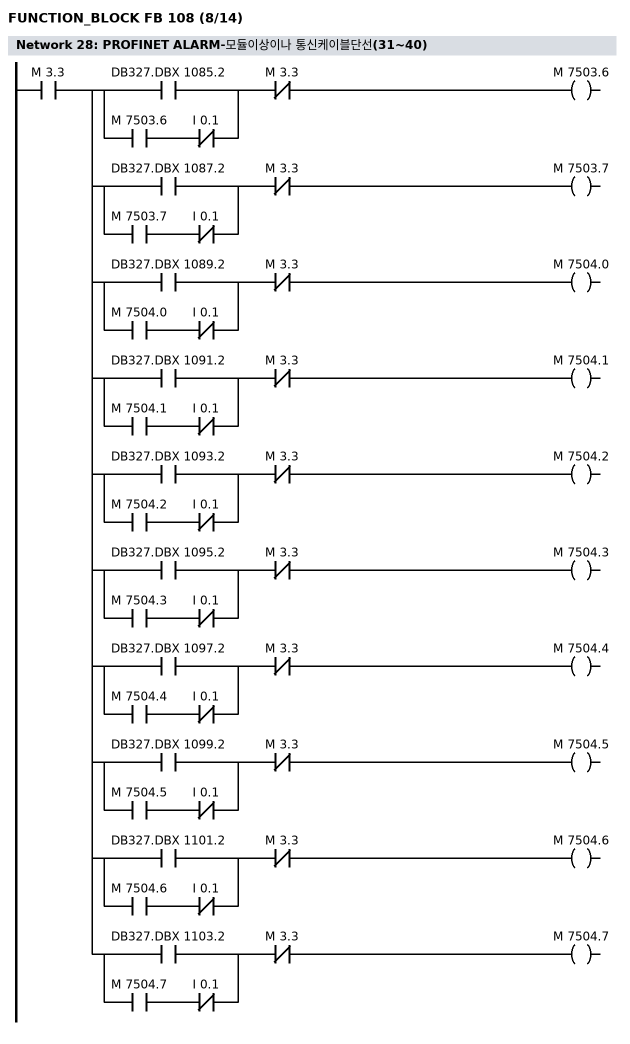
      A     M      3.3;
      =     L      0.0;
      A     L      0.0;
      A(    ;
      O     DB327.DBX 1085.2;
      O     ;
      A     M   7503.6;
      AN    I      0.1;
      )     ;
      AN    M      3.3;
      =     M   7503.6;
      A     L      0.0;
      A(    ;
      O     DB327.DBX 1087.2;
      O     ;
      A     M   7503.7;
      AN    I      0.1;
      )     ;
      AN    M      3.3;
      =     M   7503.7;
      A     L      0.0;
      A(    ;
      O     DB327.DBX 1089.2;
      O     ;
      A     M   7504.0;
      AN    I      0.1;
      )     ;
      AN    M      3.3;
      =     M   7504.0;
      A     L      0.0;
      A(    ;
      O     DB327.DBX 1091.2;
      O     ;
      A     M   7504.1;
      AN    I      0.1;
      )     ;
      AN    M      3.3;
      =     M   7504.1;
      A     L      0.0;
      A(    ;
      O     DB327.DBX 1093.2;
      O     ;
      A     M   7504.2;
      AN    I      0.1;
      )     ;
      AN    M      3.3;
      =     M   7504.2;
      A     L      0.0;
      A(    ;
      O     DB327.DBX 1095.2;
      O     ;
      A     M   7504.3;
      AN    I      0.1;
      )     ;
      AN    M      3.3;
      =     M   7504.3;
      A     L      0.0;
      A(    ;
      O     DB327.DBX 1097.2;
      O     ;
      A     M   7504.4;
      AN    I      0.1;
      )     ;
      AN    M      3.3;
      =     M   7504.4;
      A     L      0.0;
      A(    ;
      O     DB327.DBX 1099.2;
      O     ;
      A     M   7504.5;
      AN    I      0.1;
      )     ;
      AN    M      3.3;
      =     M   7504.5;
      A     L      0.0;
      A(    ;
      O     DB327.DBX 1101.2;
      O     ;
      A     M   7504.6;
      AN    I      0.1;
      )     ;
      AN    M      3.3;
      =     M   7504.6;
      A     L      0.0;
      A(    ;
      O     DB327.DBX 1103.2;
      O     ;
      A     M   7504.7;
      AN    I      0.1;
      )     ;
      AN    M      3.3;
      =     M   7504.7;
NETWORK
TITLE =PROFINET ALARM-모듈이상이나 통신케이블단선(150~159)
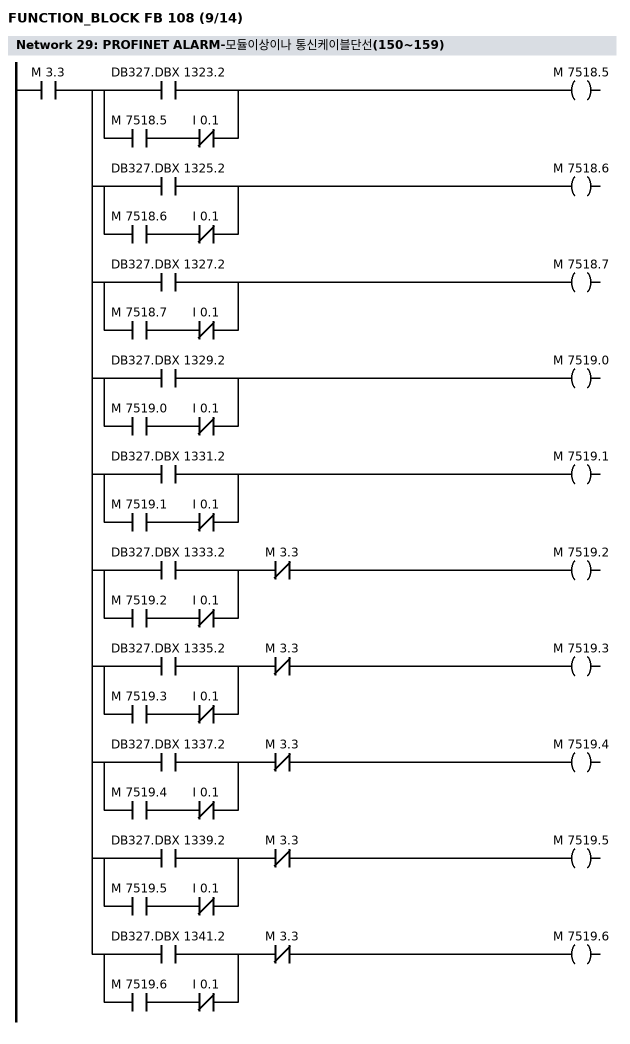

      A     M      3.3;
      =     L      0.0;
      A     L      0.0;
      A(    ;
      O     DB327.DBX 1323.2;
      O     ;
      A     M   7518.5;
      AN    I      0.1;
      )     ;
      =     M   7518.5;
      A     L      0.0;
      A(    ;
      O     DB327.DBX 1325.2;
      O     ;
      A     M   7518.6;
      AN    I      0.1;
      )     ;
      =     M   7518.6;
      A     L      0.0;
      A(    ;
      O     DB327.DBX 1327.2;
      O     ;
      A     M   7518.7;
      AN    I      0.1;
      )     ;
      =     M   7518.7;
      A     L      0.0;
      A(    ;
      O     DB327.DBX 1329.2;
      O     ;
      A     M   7519.0;
      AN    I      0.1;
      )     ;
      =     M   7519.0;
      A     L      0.0;
      A(    ;
      O     DB327.DBX 1331.2;
      O     ;
      A     M   7519.1;
      AN    I      0.1;
      )     ;
      =     M   7519.1;
      A     L      0.0;
      A(    ;
      O     DB327.DBX 1333.2;
      O     ;
      A     M   7519.2;
      AN    I      0.1;
      )     ;
      AN    M      3.3;
      =     M   7519.2;
      A     L      0.0;
      A(    ;
      O     DB327.DBX 1335.2;
      O     ;
      A     M   7519.3;
      AN    I      0.1;
      )     ;
      AN    M      3.3;
      =     M   7519.3;
      A     L      0.0;
      A(    ;
      O     DB327.DBX 1337.2;
      O     ;
      A     M   7519.4;
      AN    I      0.1;
      )     ;
      AN    M      3.3;
      =     M   7519.4;
      A     L      0.0;
      A(    ;
      O     DB327.DBX 1339.2;
      O     ;
      A     M   7519.5;
      AN    I      0.1;
      )     ;
      AN    M      3.3;
      =     M   7519.5;
      A     L      0.0;
      A(    ;
      O     DB327.DBX 1341.2;
      O     ;
      A     M   7519.6;
      AN    I      0.1;
      )     ;
      AN    M      3.3;
      =     M   7519.6;
NETWORK
TITLE =PROFINET MODULE ERROR(1~10)
//
//
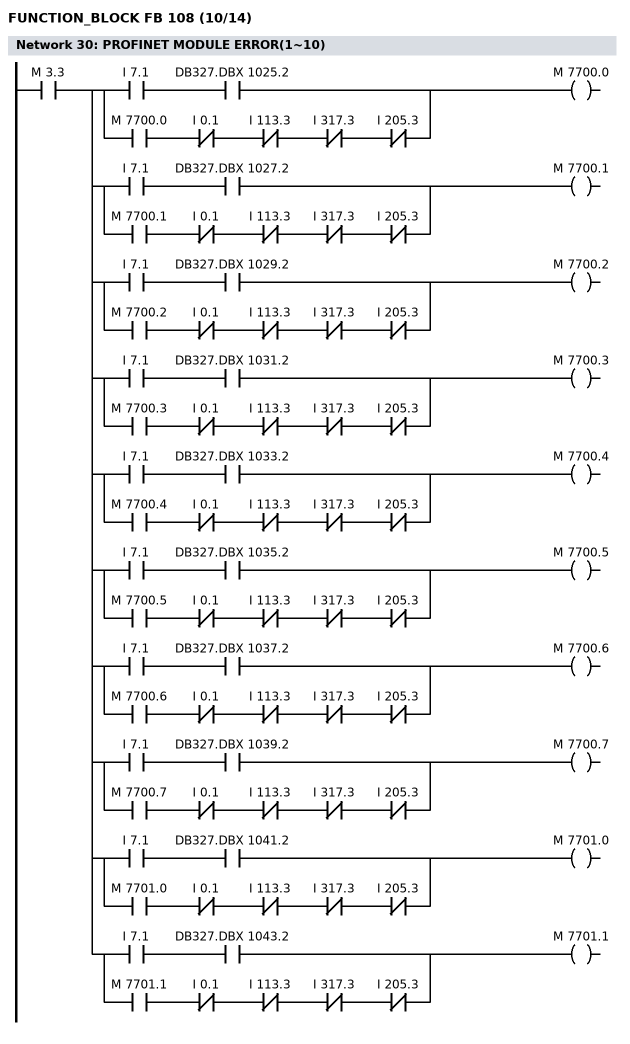
      A     M      3.3;
      =     L      0.0;
      A     L      0.0;
      A(    ;
      A     I      7.1;
      A     DB327.DBX 1025.2;
      O     ;
      A     M   7700.0;
      AN    I      0.1;
      AN    I    113.3;
      AN    I    317.3;
      AN    I    205.3;
      )     ;
      =     M   7700.0;
      A     L      0.0;
      A(    ;
      A     I      7.1;
      A     DB327.DBX 1027.2;
      O     ;
      A     M   7700.1;
      AN    I      0.1;
      AN    I    113.3;
      AN    I    317.3;
      AN    I    205.3;
      )     ;
      =     M   7700.1;
      A     L      0.0;
      A(    ;
      A     I      7.1;
      A     DB327.DBX 1029.2;
      O     ;
      A     M   7700.2;
      AN    I      0.1;
      AN    I    113.3;
      AN    I    317.3;
      AN    I    205.3;
      )     ;
      =     M   7700.2;
      A     L      0.0;
      A(    ;
      A     I      7.1;
      A     DB327.DBX 1031.2;
      O     ;
      A     M   7700.3;
      AN    I      0.1;
      AN    I    113.3;
      AN    I    317.3;
      AN    I    205.3;
      )     ;
      =     M   7700.3;
      A     L      0.0;
      A(    ;
      A     I      7.1;
      A     DB327.DBX 1033.2;
      O     ;
      A     M   7700.4;
      AN    I      0.1;
      AN    I    113.3;
      AN    I    317.3;
      AN    I    205.3;
      )     ;
      =     M   7700.4;
      A     L      0.0;
      A(    ;
      A     I      7.1;
      A     DB327.DBX 1035.2;
      O     ;
      A     M   7700.5;
      AN    I      0.1;
      AN    I    113.3;
      AN    I    317.3;
      AN    I    205.3;
      )     ;
      =     M   7700.5;
      A     L      0.0;
      A(    ;
      A     I      7.1;
      A     DB327.DBX 1037.2;
      O     ;
      A     M   7700.6;
      AN    I      0.1;
      AN    I    113.3;
      AN    I    317.3;
      AN    I    205.3;
      )     ;
      =     M   7700.6;
      A     L      0.0;
      A(    ;
      A     I      7.1;
      A     DB327.DBX 1039.2;
      O     ;
      A     M   7700.7;
      AN    I      0.1;
      AN    I    113.3;
      AN    I    317.3;
      AN    I    205.3;
      )     ;
      =     M   7700.7;
      A     L      0.0;
      A(    ;
      A     I      7.1;
      A     DB327.DBX 1041.2;
      O     ;
      A     M   7701.0;
      AN    I      0.1;
      AN    I    113.3;
      AN    I    317.3;
      AN    I    205.3;
      )     ;
      =     M   7701.0;
      A     L      0.0;
      A(    ;
      A     I      7.1;
      A     DB327.DBX 1043.2;
      O     ;
      A     M   7701.1;
      AN    I      0.1;
      AN    I    113.3;
      AN    I    317.3;
      AN    I    205.3;
      )     ;
      =     M   7701.1;
NETWORK
TITLE =PROFINET MODULE ERROR(11~20)
//
//
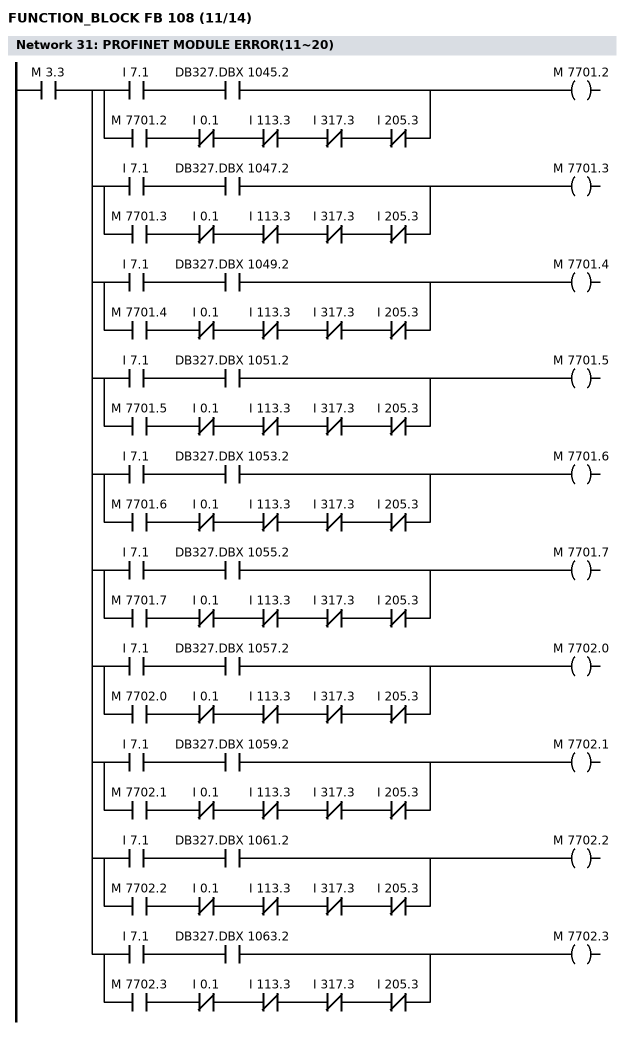
      A     M      3.3;
      =     L      0.0;
      A     L      0.0;
      A(    ;
      A     I      7.1;
      A     DB327.DBX 1045.2;
      O     ;
      A     M   7701.2;
      AN    I      0.1;
      AN    I    113.3;
      AN    I    317.3;
      AN    I    205.3;
      )     ;
      =     M   7701.2;
      A     L      0.0;
      A(    ;
      A     I      7.1;
      A     DB327.DBX 1047.2;
      O     ;
      A     M   7701.3;
      AN    I      0.1;
      AN    I    113.3;
      AN    I    317.3;
      AN    I    205.3;
      )     ;
      =     M   7701.3;
      A     L      0.0;
      A(    ;
      A     I      7.1;
      A     DB327.DBX 1049.2;
      O     ;
      A     M   7701.4;
      AN    I      0.1;
      AN    I    113.3;
      AN    I    317.3;
      AN    I    205.3;
      )     ;
      =     M   7701.4;
      A     L      0.0;
      A(    ;
      A     I      7.1;
      A     DB327.DBX 1051.2;
      O     ;
      A     M   7701.5;
      AN    I      0.1;
      AN    I    113.3;
      AN    I    317.3;
      AN    I    205.3;
      )     ;
      =     M   7701.5;
      A     L      0.0;
      A(    ;
      A     I      7.1;
      A     DB327.DBX 1053.2;
      O     ;
      A     M   7701.6;
      AN    I      0.1;
      AN    I    113.3;
      AN    I    317.3;
      AN    I    205.3;
      )     ;
      =     M   7701.6;
      A     L      0.0;
      A(    ;
      A     I      7.1;
      A     DB327.DBX 1055.2;
      O     ;
      A     M   7701.7;
      AN    I      0.1;
      AN    I    113.3;
      AN    I    317.3;
      AN    I    205.3;
      )     ;
      =     M   7701.7;
      A     L      0.0;
      A(    ;
      A     I      7.1;
      A     DB327.DBX 1057.2;
      O     ;
      A     M   7702.0;
      AN    I      0.1;
      AN    I    113.3;
      AN    I    317.3;
      AN    I    205.3;
      )     ;
      =     M   7702.0;
      A     L      0.0;
      A(    ;
      A     I      7.1;
      A     DB327.DBX 1059.2;
      O     ;
      A     M   7702.1;
      AN    I      0.1;
      AN    I    113.3;
      AN    I    317.3;
      AN    I    205.3;
      )     ;
      =     M   7702.1;
      A     L      0.0;
      A(    ;
      A     I      7.1;
      A     DB327.DBX 1061.2;
      O     ;
      A     M   7702.2;
      AN    I      0.1;
      AN    I    113.3;
      AN    I    317.3;
      AN    I    205.3;
      )     ;
      =     M   7702.2;
      A     L      0.0;
      A(    ;
      A     I      7.1;
      A     DB327.DBX 1063.2;
      O     ;
      A     M   7702.3;
      AN    I      0.1;
      AN    I    113.3;
      AN    I    317.3;
      AN    I    205.3;
      )     ;
      =     M   7702.3;
NETWORK
TITLE =PROFINET MODULE ERROR(21~30)
//
//
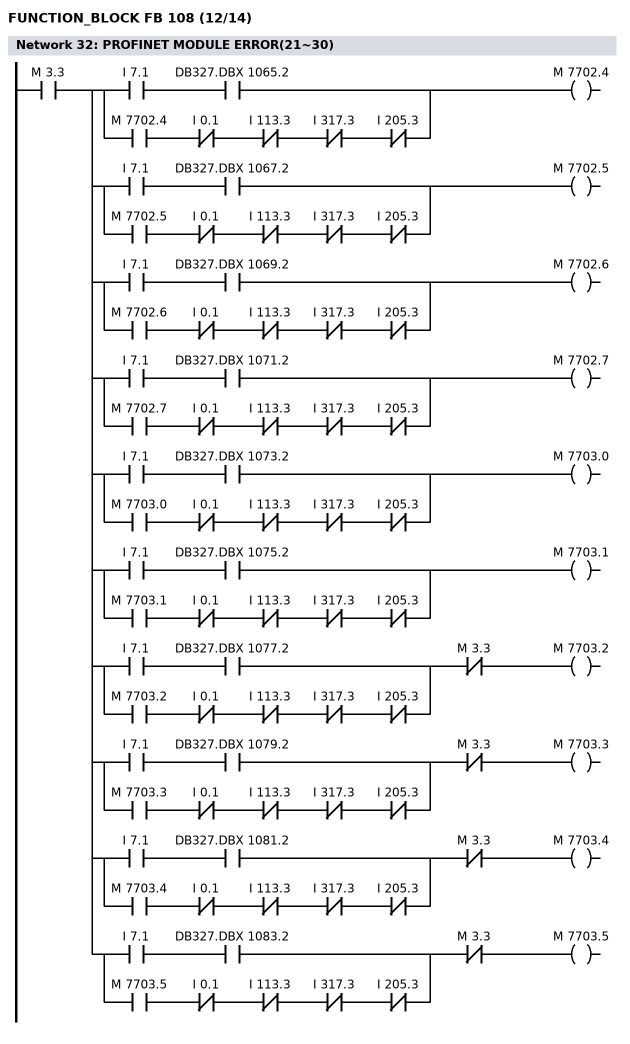
      A     M      3.3;
      =     L      0.0;
      A     L      0.0;
      A(    ;
      A     I      7.1;
      A     DB327.DBX 1065.2;
      O     ;
      A     M   7702.4;
      AN    I      0.1;
      AN    I    113.3;
      AN    I    317.3;
      AN    I    205.3;
      )     ;
      =     M   7702.4;
      A     L      0.0;
      A(    ;
      A     I      7.1;
      A     DB327.DBX 1067.2;
      O     ;
      A     M   7702.5;
      AN    I      0.1;
      AN    I    113.3;
      AN    I    317.3;
      AN    I    205.3;
      )     ;
      =     M   7702.5;
      A     L      0.0;
      A(    ;
      A     I      7.1;
      A     DB327.DBX 1069.2;
      O     ;
      A     M   7702.6;
      AN    I      0.1;
      AN    I    113.3;
      AN    I    317.3;
      AN    I    205.3;
      )     ;
      =     M   7702.6;
      A     L      0.0;
      A(    ;
      A     I      7.1;
      A     DB327.DBX 1071.2;
      O     ;
      A     M   7702.7;
      AN    I      0.1;
      AN    I    113.3;
      AN    I    317.3;
      AN    I    205.3;
      )     ;
      =     M   7702.7;
      A     L      0.0;
      A(    ;
      A     I      7.1;
      A     DB327.DBX 1073.2;
      O     ;
      A     M   7703.0;
      AN    I      0.1;
      AN    I    113.3;
      AN    I    317.3;
      AN    I    205.3;
      )     ;
      =     M   7703.0;
      A     L      0.0;
      A(    ;
      A     I      7.1;
      A     DB327.DBX 1075.2;
      O     ;
      A     M   7703.1;
      AN    I      0.1;
      AN    I    113.3;
      AN    I    317.3;
      AN    I    205.3;
      )     ;
      =     M   7703.1;
      A     L      0.0;
      A(    ;
      A     I      7.1;
      A     DB327.DBX 1077.2;
      O     ;
      A     M   7703.2;
      AN    I      0.1;
      AN    I    113.3;
      AN    I    317.3;
      AN    I    205.3;
      )     ;
      AN    M      3.3;
      =     M   7703.2;
      A     L      0.0;
      A(    ;
      A     I      7.1;
      A     DB327.DBX 1079.2;
      O     ;
      A     M   7703.3;
      AN    I      0.1;
      AN    I    113.3;
      AN    I    317.3;
      AN    I    205.3;
      )     ;
      AN    M      3.3;
      =     M   7703.3;
      A     L      0.0;
      A(    ;
      A     I      7.1;
      A     DB327.DBX 1081.2;
      O     ;
      A     M   7703.4;
      AN    I      0.1;
      AN    I    113.3;
      AN    I    317.3;
      AN    I    205.3;
      )     ;
      AN    M      3.3;
      =     M   7703.4;
      A     L      0.0;
      A(    ;
      A     I      7.1;
      A     DB327.DBX 1083.2;
      O     ;
      A     M   7703.5;
      AN    I      0.1;
      AN    I    113.3;
      AN    I    317.3;
      AN    I    205.3;
      )     ;
      AN    M      3.3;
      =     M   7703.5;
NETWORK
TITLE =PROFINET MODULE ERROR(31~40)
//
//
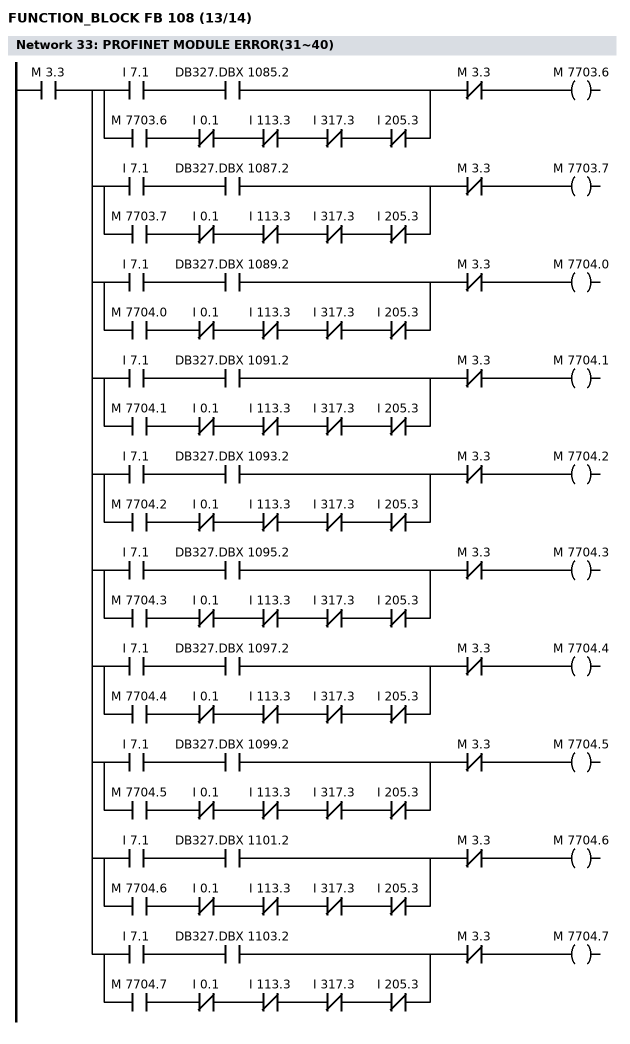
      A     M      3.3;
      =     L      0.0;
      A     L      0.0;
      A(    ;
      A     I      7.1;
      A     DB327.DBX 1085.2;
      O     ;
      A     M   7703.6;
      AN    I      0.1;
      AN    I    113.3;
      AN    I    317.3;
      AN    I    205.3;
      )     ;
      AN    M      3.3;
      =     M   7703.6;
      A     L      0.0;
      A(    ;
      A     I      7.1;
      A     DB327.DBX 1087.2;
      O     ;
      A     M   7703.7;
      AN    I      0.1;
      AN    I    113.3;
      AN    I    317.3;
      AN    I    205.3;
      )     ;
      AN    M      3.3;
      =     M   7703.7;
      A     L      0.0;
      A(    ;
      A     I      7.1;
      A     DB327.DBX 1089.2;
      O     ;
      A     M   7704.0;
      AN    I      0.1;
      AN    I    113.3;
      AN    I    317.3;
      AN    I    205.3;
      )     ;
      AN    M      3.3;
      =     M   7704.0;
      A     L      0.0;
      A(    ;
      A     I      7.1;
      A     DB327.DBX 1091.2;
      O     ;
      A     M   7704.1;
      AN    I      0.1;
      AN    I    113.3;
      AN    I    317.3;
      AN    I    205.3;
      )     ;
      AN    M      3.3;
      =     M   7704.1;
      A     L      0.0;
      A(    ;
      A     I      7.1;
      A     DB327.DBX 1093.2;
      O     ;
      A     M   7704.2;
      AN    I      0.1;
      AN    I    113.3;
      AN    I    317.3;
      AN    I    205.3;
      )     ;
      AN    M      3.3;
      =     M   7704.2;
      A     L      0.0;
      A(    ;
      A     I      7.1;
      A     DB327.DBX 1095.2;
      O     ;
      A     M   7704.3;
      AN    I      0.1;
      AN    I    113.3;
      AN    I    317.3;
      AN    I    205.3;
      )     ;
      AN    M      3.3;
      =     M   7704.3;
      A     L      0.0;
      A(    ;
      A     I      7.1;
      A     DB327.DBX 1097.2;
      O     ;
      A     M   7704.4;
      AN    I      0.1;
      AN    I    113.3;
      AN    I    317.3;
      AN    I    205.3;
      )     ;
      AN    M      3.3;
      =     M   7704.4;
      A     L      0.0;
      A(    ;
      A     I      7.1;
      A     DB327.DBX 1099.2;
      O     ;
      A     M   7704.5;
      AN    I      0.1;
      AN    I    113.3;
      AN    I    317.3;
      AN    I    205.3;
      )     ;
      AN    M      3.3;
      =     M   7704.5;
      A     L      0.0;
      A(    ;
      A     I      7.1;
      A     DB327.DBX 1101.2;
      O     ;
      A     M   7704.6;
      AN    I      0.1;
      AN    I    113.3;
      AN    I    317.3;
      AN    I    205.3;
      )     ;
      AN    M      3.3;
      =     M   7704.6;
      A     L      0.0;
      A(    ;
      A     I      7.1;
      A     DB327.DBX 1103.2;
      O     ;
      A     M   7704.7;
      AN    I      0.1;
      AN    I    113.3;
      AN    I    317.3;
      AN    I    205.3;
      )     ;
      AN    M      3.3;
      =     M   7704.7;
NETWORK
TITLE =PROFINET MODULE ERROR(150~159)
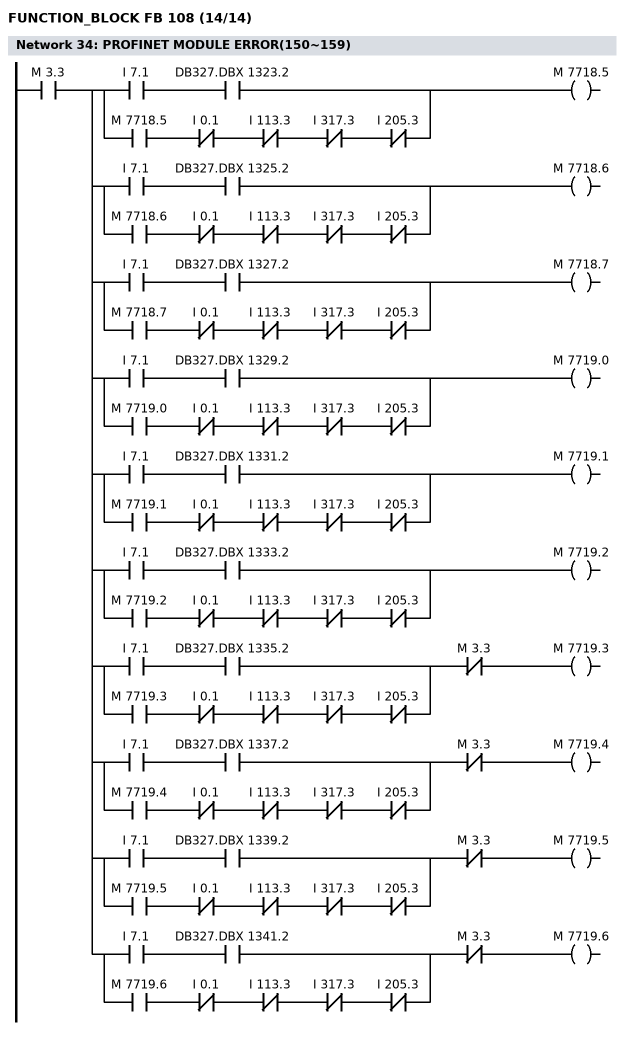

      A     M      3.3;
      =     L      0.0;
      A     L      0.0;
      A(    ;
      A     I      7.1;
      A     DB327.DBX 1323.2;
      O     ;
      A     M   7718.5;
      AN    I      0.1;
      AN    I    113.3;
      AN    I    317.3;
      AN    I    205.3;
      )     ;
      =     M   7718.5;
      A     L      0.0;
      A(    ;
      A     I      7.1;
      A     DB327.DBX 1325.2;
      O     ;
      A     M   7718.6;
      AN    I      0.1;
      AN    I    113.3;
      AN    I    317.3;
      AN    I    205.3;
      )     ;
      =     M   7718.6;
      A     L      0.0;
      A(    ;
      A     I      7.1;
      A     DB327.DBX 1327.2;
      O     ;
      A     M   7718.7;
      AN    I      0.1;
      AN    I    113.3;
      AN    I    317.3;
      AN    I    205.3;
      )     ;
      =     M   7718.7;
      A     L      0.0;
      A(    ;
      A     I      7.1;
      A     DB327.DBX 1329.2;
      O     ;
      A     M   7719.0;
      AN    I      0.1;
      AN    I    113.3;
      AN    I    317.3;
      AN    I    205.3;
      )     ;
      =     M   7719.0;
      A     L      0.0;
      A(    ;
      A     I      7.1;
      A     DB327.DBX 1331.2;
      O     ;
      A     M   7719.1;
      AN    I      0.1;
      AN    I    113.3;
      AN    I    317.3;
      AN    I    205.3;
      )     ;
      =     M   7719.1;
      A     L      0.0;
      A(    ;
      A     I      7.1;
      A     DB327.DBX 1333.2;
      O     ;
      A     M   7719.2;
      AN    I      0.1;
      AN    I    113.3;
      AN    I    317.3;
      AN    I    205.3;
      )     ;
      =     M   7719.2;
      A     L      0.0;
      A(    ;
      A     I      7.1;
      A     DB327.DBX 1335.2;
      O     ;
      A     M   7719.3;
      AN    I      0.1;
      AN    I    113.3;
      AN    I    317.3;
      AN    I    205.3;
      )     ;
      AN    M      3.3;
      =     M   7719.3;
      A     L      0.0;
      A(    ;
      A     I      7.1;
      A     DB327.DBX 1337.2;
      O     ;
      A     M   7719.4;
      AN    I      0.1;
      AN    I    113.3;
      AN    I    317.3;
      AN    I    205.3;
      )     ;
      AN    M      3.3;
      =     M   7719.4;
      A     L      0.0;
      A(    ;
      A     I      7.1;
      A     DB327.DBX 1339.2;
      O     ;
      A     M   7719.5;
      AN    I      0.1;
      AN    I    113.3;
      AN    I    317.3;
      AN    I    205.3;
      )     ;
      AN    M      3.3;
      =     M   7719.5;
      A     L      0.0;
      A(    ;
      A     I      7.1;
      A     DB327.DBX 1341.2;
      O     ;
      A     M   7719.6;
      AN    I      0.1;
      AN    I    113.3;
      AN    I    317.3;
      AN    I    205.3;
      )     ;
      AN    M      3.3;
      =     M   7719.6;
END_FUNCTION_BLOCK

DATA_BLOCK DB 108
TITLE =
VERSION : 0.0

 FB 108
BEGIN
END_DATA_BLOCK

FUNCTION FC 108 : VOID
TITLE =
VERSION : 0.1

BEGIN
NETWORK
TITLE =
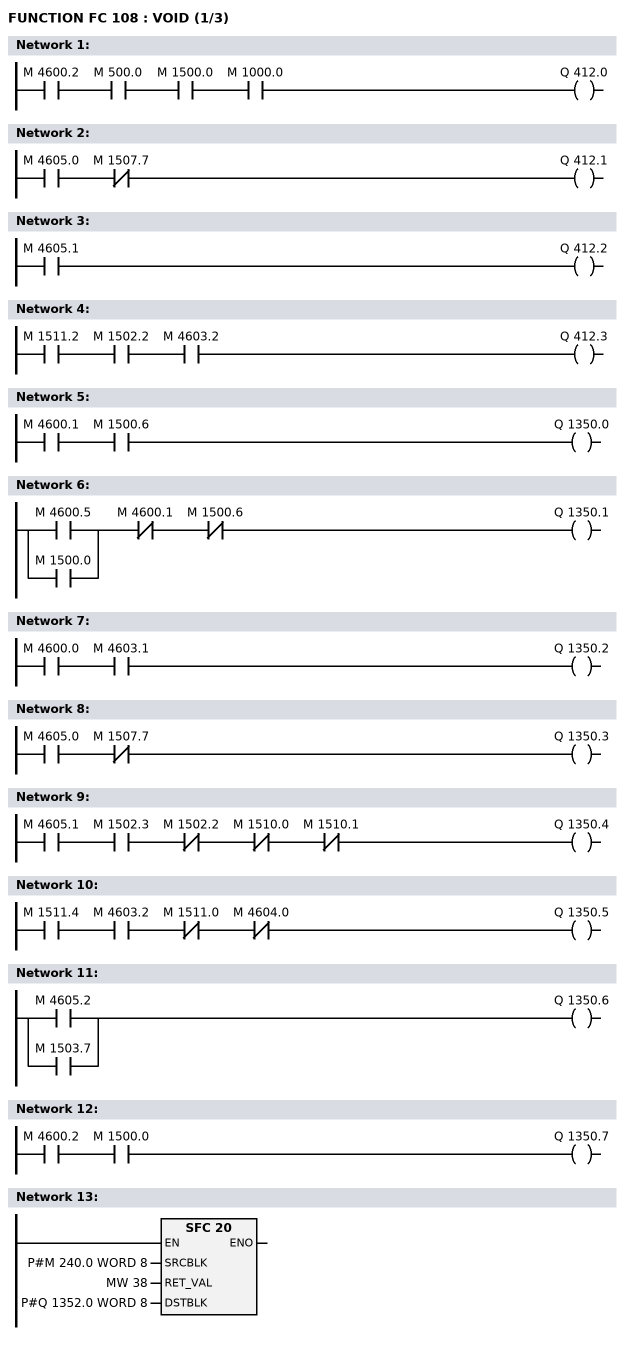

      A     M   4600.2;
      A     M    500.0;
      A     M   1500.0;
      A     M   1000.0;
      =     Q    412.0;
NETWORK
TITLE =

      A     M   4605.0;
      AN    M   1507.7;
      =     Q    412.1;
NETWORK
TITLE =

      A     M   4605.1;
      =     Q    412.2;
NETWORK
TITLE =

      A     M   1511.2;
      A     M   1502.2;
      A     M   4603.2;
      =     Q    412.3;
NETWORK
TITLE =

      A     M   4600.1;
      A     M   1500.6;
      =     Q   1350.0;
NETWORK
TITLE =

      A(    ;
      O     M   4600.5;
      O     M   1500.0;
      )     ;
      AN    M   4600.1;
      AN    M   1500.6;
      =     Q   1350.1;
NETWORK
TITLE =

      A     M   4600.0;
      A     M   4603.1;
      =     Q   1350.2;
NETWORK
TITLE =

      A     M   4605.0;
      AN    M   1507.7;
      =     Q   1350.3;
NETWORK
TITLE =

      A     M   4605.1;
      A     M   1502.3;
      AN    M   1502.2;
      AN    M   1510.0;
      AN    M   1510.1;
      =     Q   1350.4;
NETWORK
TITLE =

      A     M   1511.4;
      A     M   4603.2;
      AN    M   1511.0;
      AN    M   4604.0;
      =     Q   1350.5;
NETWORK
TITLE =

      O     M   4605.2;
      O     M   1503.7;
      =     Q   1350.6;
NETWORK
TITLE =

      A     M   4600.2;
      A     M   1500.0;
      =     Q   1350.7;
NETWORK
TITLE =

      CALL SFC   20 (
           SRCBLK                   := P#M 240.0 WORD 8,
           RET_VAL                  := MW    38,
           DSTBLK                   := P#Q 1352.0 WORD 8);
      NOP   0;
NETWORK
TITLE =
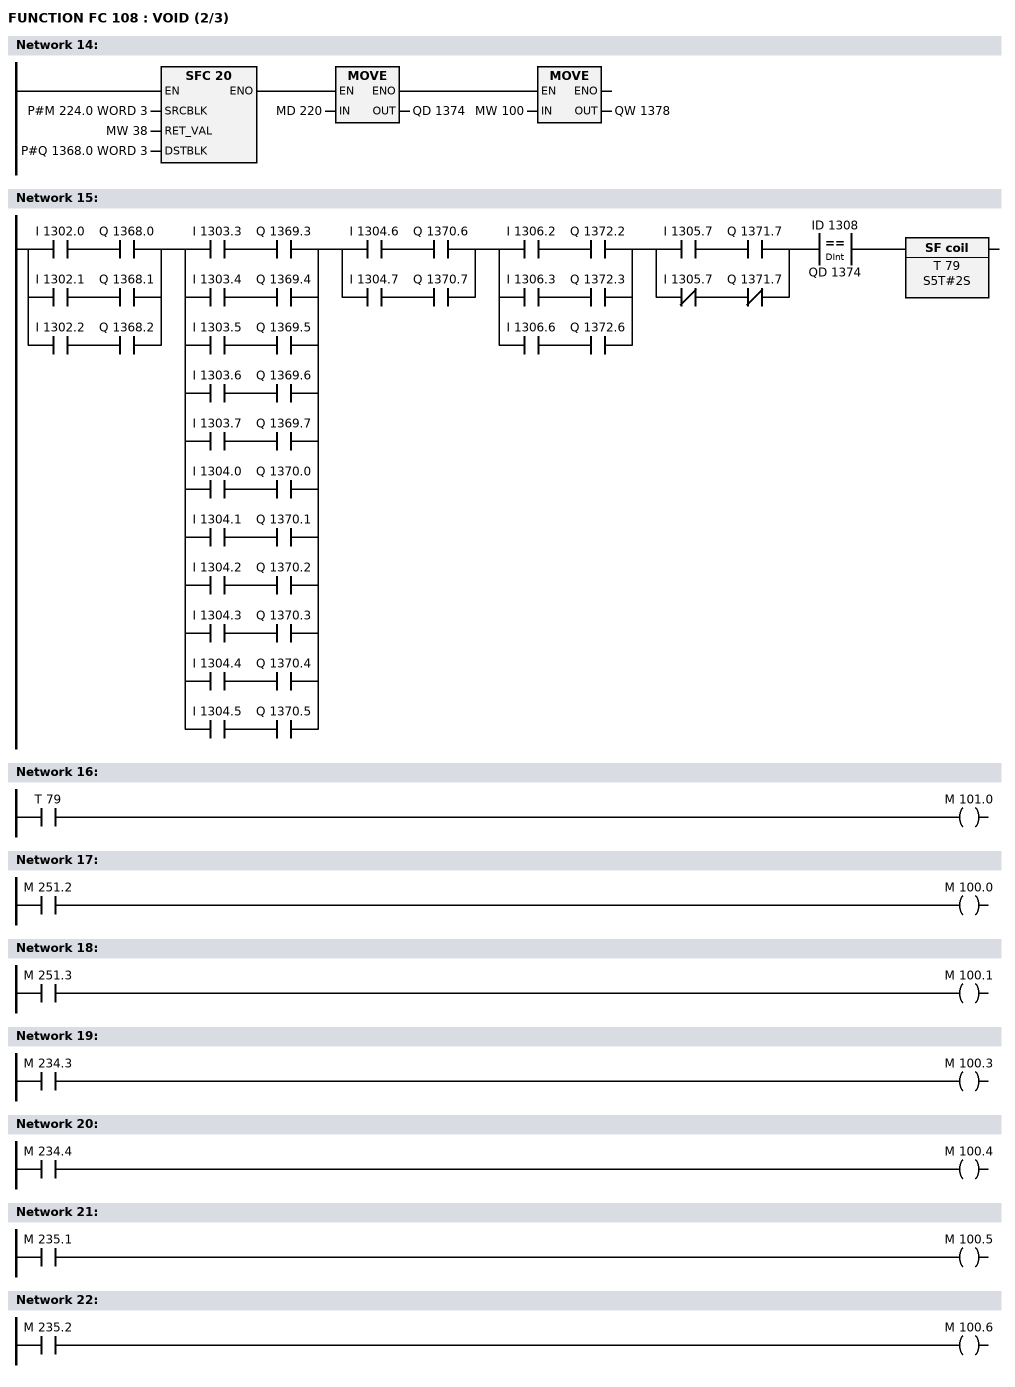

      A(    ;
      A(    ;
      CALL SFC   20 (
           SRCBLK                   := P#M 224.0 WORD 3,
           RET_VAL                  := MW    38,
           DSTBLK                   := P#Q 1368.0 WORD 3);
      A     BR;
      )     ;
      JNB   _001;
      L     MD   220;
      T     QD  1374;
      SET   ;
      SAVE  ;
      CLR   ;
_001: A     BR;
      )     ;
      JNB   _002;
      L     MW   100;
      T     QW  1378;
_002: NOP   0;
NETWORK
TITLE =

      A(    ;
      A     I   1302.0;
      A     Q   1368.0;
      O     ;
      A     I   1302.1;
      A     Q   1368.1;
      O     ;
      A     I   1302.2;
      A     Q   1368.2;
      )     ;
      A(    ;
      A     I   1303.3;
      A     Q   1369.3;
      O     ;
      A     I   1303.4;
      A     Q   1369.4;
      O     ;
      A     I   1303.5;
      A     Q   1369.5;
      O     ;
      A     I   1303.6;
      A     Q   1369.6;
      O     ;
      A     I   1303.7;
      A     Q   1369.7;
      O     ;
      A     I   1304.0;
      A     Q   1370.0;
      O     ;
      A     I   1304.1;
      A     Q   1370.1;
      O     ;
      A     I   1304.2;
      A     Q   1370.2;
      O     ;
      A     I   1304.3;
      A     Q   1370.3;
      O     ;
      A     I   1304.4;
      A     Q   1370.4;
      O     ;
      A     I   1304.5;
      A     Q   1370.5;
      )     ;
      A(    ;
      A     I   1304.6;
      A     Q   1370.6;
      O     ;
      A     I   1304.7;
      A     Q   1370.7;
      )     ;
      A(    ;
      A     I   1306.2;
      A     Q   1372.2;
      O     ;
      A     I   1306.3;
      A     Q   1372.3;
      O     ;
      A     I   1306.6;
      A     Q   1372.6;
      )     ;
      A(    ;
      A     I   1305.7;
      A     Q   1371.7;
      O     ;
      AN    I   1305.7;
      AN    Q   1371.7;
      )     ;
      A(    ;
      L     ID  1308;
      L     QD  1374;
      ==D   ;
      )     ;
      L     S5T#2S;
      SF    T     79;
NETWORK
TITLE =

      A     T     79;
      =     M    101.0;
NETWORK
TITLE =

      A     M    251.2;
      =     M    100.0;
NETWORK
TITLE =

      A     M    251.3;
      =     M    100.1;
NETWORK
TITLE =

      A     M    234.3;
      =     M    100.3;
NETWORK
TITLE =

      A     M    234.4;
      =     M    100.4;
NETWORK
TITLE =

      A     M    235.1;
      =     M    100.5;
NETWORK
TITLE =

      A     M    235.2;
      =     M    100.6;
NETWORK
TITLE =
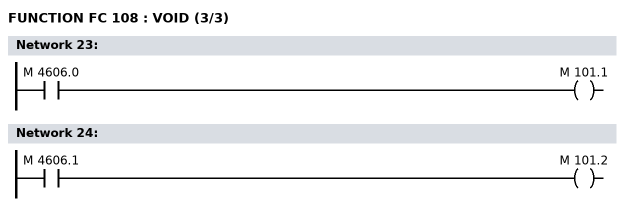

      A     M   4606.0;
      =     M    101.1;
NETWORK
TITLE =

      A     M   4606.1;
      =     M    101.2;
END_FUNCTION

FUNCTION_BLOCK FB 110
TITLE =
VERSION : 0.1


VAR
  S_OUT_TRV_MODE : FB 402;
END_VAR
BEGIN
NETWORK
TITLE =
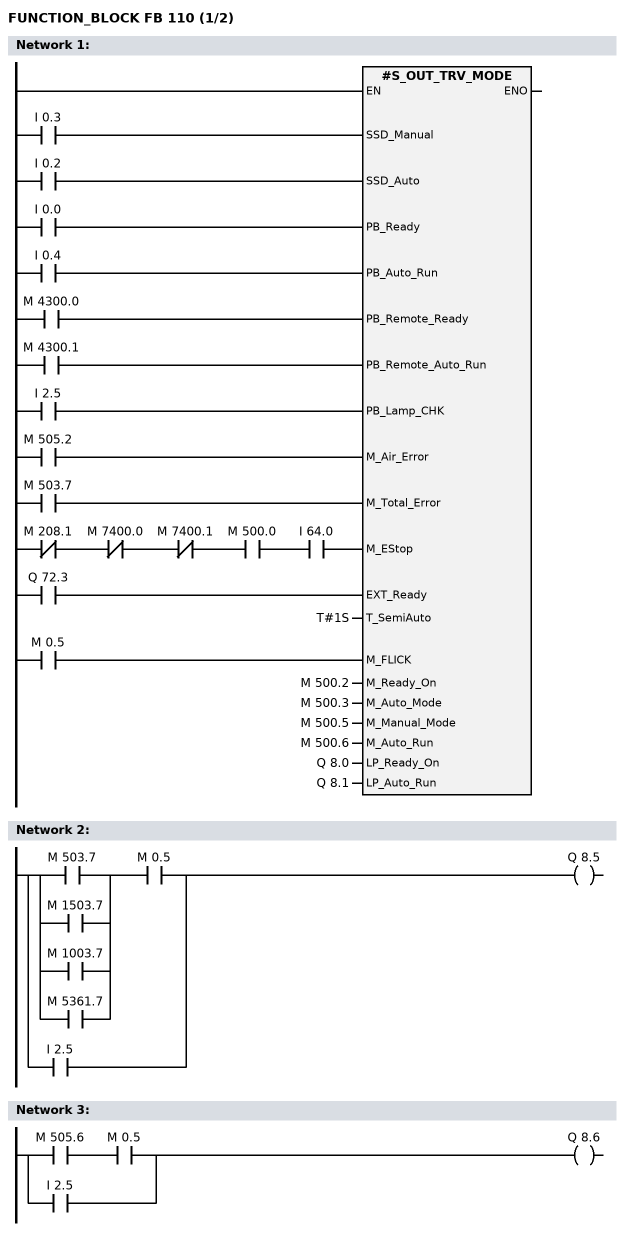

      A     I      0.3;
      =     L      0.0;
      BLD   103;
      A     I      0.2;
      =     L      0.1;
      BLD   103;
      A     I      0.0;
      =     L      0.2;
      BLD   103;
      A     I      0.4;
      =     L      0.3;
      BLD   103;
      A     M   4300.0;
      =     L      0.4;
      BLD   103;
      A     M   4300.1;
      =     L      0.5;
      BLD   103;
      A     I      2.5;
      =     L      0.6;
      BLD   103;
      A     M    505.2;
      =     L      0.7;
      BLD   103;
      A     M    503.7;
      =     L      1.1;
      BLD   103;
      AN    M    208.1;
      AN    M   7400.0;
      AN    M   7400.1;
      A     M    500.0;
      A     I     64.0;
      =     L      1.2;
      BLD   103;
      A     Q     72.3;
      =     L      1.3;
      BLD   103;
      A     M      0.5;
      =     L      1.5;
      BLD   103;
      CALL #S_OUT_TRV_MODE (
           SSD_Manual               := L      0.0,
           SSD_Auto                 := L      0.1,
           PB_Ready                 := L      0.2,
           PB_Auto_Run              := L      0.3,
           PB_Remote_Ready          := L      0.4,
           PB_Remote_Auto_Run       := L      0.5,
           PB_Lamp_CHK              := L      0.6,
           M_Air_Error              := L      0.7,
           M_Total_Error            := L      1.1,
           M_EStop                  := L      1.2,
           EXT_Ready                := L      1.3,
           T_SemiAuto               := T#1S,
           M_FLICK                  := L      1.5,
           M_Ready_On               := M    500.2,
           M_Auto_Mode              := M    500.3,
           M_Manual_Mode            := M    500.5,
           M_Auto_Run               := M    500.6,
           LP_Ready_On              := Q      8.0,
           LP_Auto_Run              := Q      8.1);
      NOP   0;
NETWORK
TITLE =

      A(    ;
      O     M    503.7;
      O     M   1503.7;
      O     M   1003.7;
      O     M   5361.7;
      )     ;
      A     M      0.5;
      O     I      2.5;
      =     Q      8.5;
NETWORK
TITLE =

      A     M    505.6;
      A     M      0.5;
      O     I      2.5;
      =     Q      8.6;
NETWORK
TITLE =
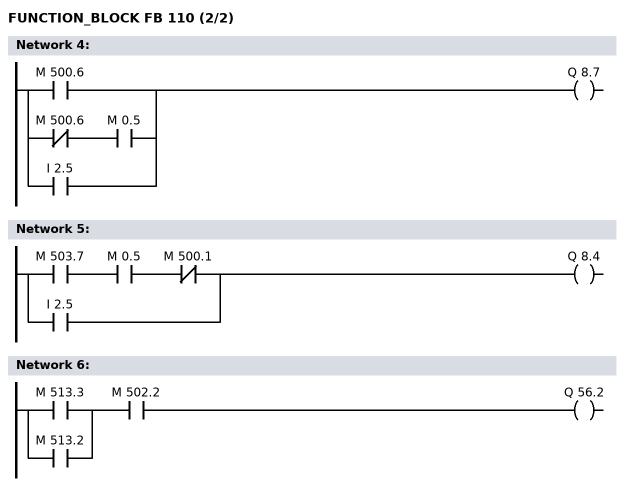

      O     M    500.6;
      O     ;
      AN    M    500.6;
      A     M      0.5;
      O     I      2.5;
      =     Q      8.7;
NETWORK
TITLE =

      A     M    503.7;
      A     M      0.5;
      AN    M    500.1;
      O     I      2.5;
      =     Q      8.4;
NETWORK
TITLE =

      A(    ;
      O     M    513.3;
      O     M    513.2;
      )     ;
      A     M    502.2;
      =     Q     56.2;
END_FUNCTION_BLOCK

DATA_BLOCK DB 110
TITLE =
VERSION : 0.0

 FB 110
BEGIN
   S_OUT_TRV_MODE.SSD_Manual := FALSE;
   S_OUT_TRV_MODE.SSD_Auto := FALSE;
   S_OUT_TRV_MODE.PB_Ready := FALSE;
   S_OUT_TRV_MODE.PB_Auto_Run := FALSE;
   S_OUT_TRV_MODE.PB_Remote_Ready := FALSE;
   S_OUT_TRV_MODE.PB_Remote_Auto_Run := FALSE;
   S_OUT_TRV_MODE.PB_Lamp_CHK := FALSE;
   S_OUT_TRV_MODE.M_Air_Error := FALSE;
   S_OUT_TRV_MODE.M_Water_Error := FALSE;
   S_OUT_TRV_MODE.M_Total_Error := FALSE;
   S_OUT_TRV_MODE.M_EStop := FALSE;
   S_OUT_TRV_MODE.EXT_Ready := FALSE;
   S_OUT_TRV_MODE.EXT_Auto := FALSE;
   S_OUT_TRV_MODE.T_SemiAuto := T#0MS;
   S_OUT_TRV_MODE.M_FLICK := FALSE;
   S_OUT_TRV_MODE.M_Ready_On := FALSE;
   S_OUT_TRV_MODE.M_Auto_Mode := FALSE;
   S_OUT_TRV_MODE.M_SemiAuto_Mode := FALSE;
   S_OUT_TRV_MODE.M_Manual_Mode := FALSE;
   S_OUT_TRV_MODE.M_Auto_Run := FALSE;
   S_OUT_TRV_MODE.LP_Ready_On := FALSE;
   S_OUT_TRV_MODE.LP_Auto_Run := FALSE;
   S_OUT_TRV_MODE.AUTO_MODE_DELAY.IN := FALSE;
   S_OUT_TRV_MODE.AUTO_MODE_DELAY.PT := T#0MS;
   S_OUT_TRV_MODE.AUTO_MODE_DELAY.Q := FALSE;
   S_OUT_TRV_MODE.AUTO_MODE_DELAY.ET := T#0MS;
   S_OUT_TRV_MODE.AUTO_MODE_DELAY.STATE := B#16#0;
   S_OUT_TRV_MODE.AUTO_MODE_DELAY.STIME := T#0MS;
   S_OUT_TRV_MODE.AUTO_MODE_DELAY.ATIME := T#0MS;
   S_OUT_TRV_MODE.SEMI_AUTO_DELAY.IN := FALSE;
   S_OUT_TRV_MODE.SEMI_AUTO_DELAY.PT := T#0MS;
   S_OUT_TRV_MODE.SEMI_AUTO_DELAY.Q := FALSE;
   S_OUT_TRV_MODE.SEMI_AUTO_DELAY.ET := T#0MS;
   S_OUT_TRV_MODE.SEMI_AUTO_DELAY.STATE := B#16#0;
   S_OUT_TRV_MODE.SEMI_AUTO_DELAY.STIME := T#0MS;
   S_OUT_TRV_MODE.SEMI_AUTO_DELAY.ATIME := T#0MS;
   S_OUT_TRV_MODE.MANUAL_DELAY.IN := FALSE;
   S_OUT_TRV_MODE.MANUAL_DELAY.PT := T#0MS;
   S_OUT_TRV_MODE.MANUAL_DELAY.Q := FALSE;
   S_OUT_TRV_MODE.MANUAL_DELAY.ET := T#0MS;
   S_OUT_TRV_MODE.MANUAL_DELAY.STATE := B#16#0;
   S_OUT_TRV_MODE.MANUAL_DELAY.STIME := T#0MS;
   S_OUT_TRV_MODE.MANUAL_DELAY.ATIME := T#0MS;
END_DATA_BLOCK

FUNCTION FC 110 : VOID
TITLE =
VERSION : 0.1

BEGIN
NETWORK
TITLE =
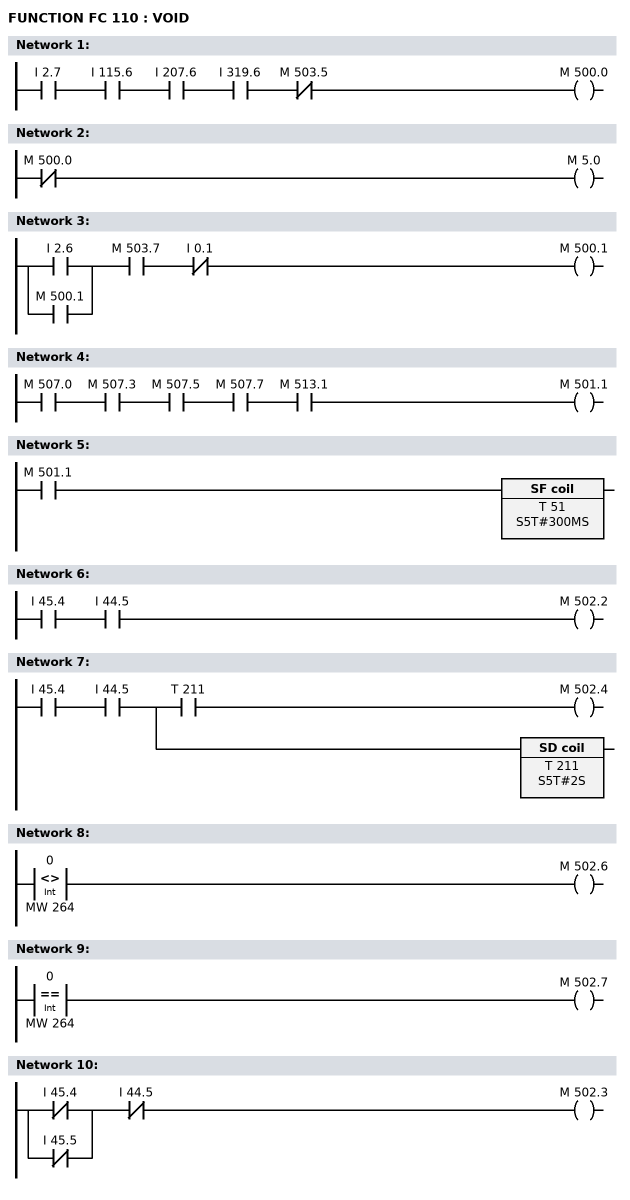

      A     I      2.7;
      A     I    115.6;
      A     I    207.6;
      A     I    319.6;
      AN    M    503.5;
      =     M    500.0;
NETWORK
TITLE =

      AN    M    500.0;
      =     M      5.0;
NETWORK
TITLE =

      A(    ;
      O     I      2.6;
      O     M    500.1;
      )     ;
      A     M    503.7;
      AN    I      0.1;
      =     M    500.1;
NETWORK
TITLE =

      A     M    507.0;
      A     M    507.3;
      A     M    507.5;
      A     M    507.7;
      A     M    513.1;
      =     M    501.1;
NETWORK
TITLE =

      A     M    501.1;
      L     S5T#300MS;
      SF    T     51;
NETWORK
TITLE =

      A     I     45.4;
      A     I     44.5;
      =     M    502.2;
NETWORK
TITLE =

      A     I     45.4;
      A     I     44.5;
      =     L      0.0;
      A     L      0.0;
      A     T    211;
      =     M    502.4;
      A     L      0.0;
      BLD   102;
      L     S5T#2S;
      SD    T    211;
NETWORK
TITLE =

      L     0;
      L     MW   264;
      <>I   ;
      =     M    502.6;
NETWORK
TITLE =

      L     0;
      L     MW   264;
      ==I   ;
      =     M    502.7;
NETWORK
TITLE =

      A(    ;
      ON    I     45.4;
      ON    I     45.5;
      )     ;
      AN    I     44.5;
      =     M    502.3;
END_FUNCTION

FUNCTION_BLOCK FB 111
TITLE =
VERSION : 0.1


VAR
  OUT_TRV_CUSHION_B : FB 424;
  OUT_TRV_GUIDE : FB 424;
  OUT_TRV_CLAMP : FB 424;
  OUT_TRV_LIFT : FB 424;
  OUT_TRV_ELE : FB 424;
END_VAR
BEGIN
NETWORK
TITLE =
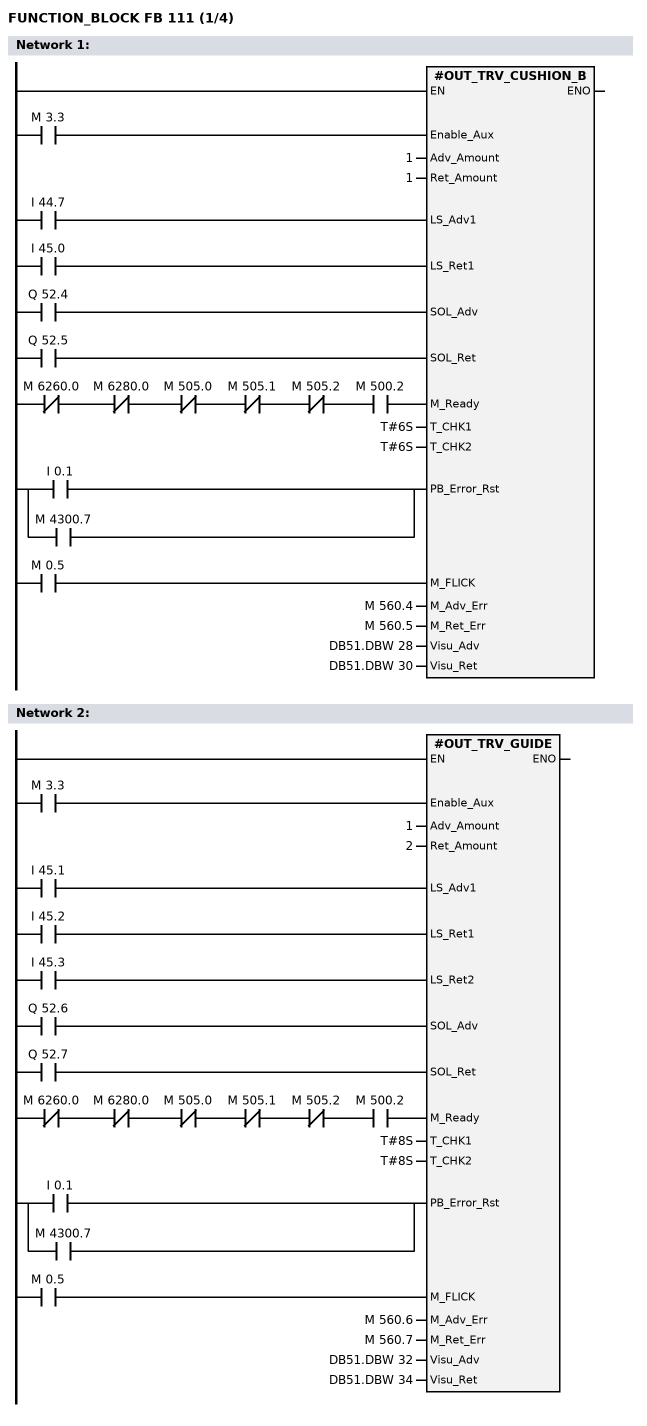

      A     M      3.3;
      =     L      0.0;
      BLD   103;
      A     I     44.7;
      =     L      0.1;
      BLD   103;
      A     I     45.0;
      =     L      0.2;
      BLD   103;
      A     Q     52.4;
      =     L      1.1;
      BLD   103;
      A     Q     52.5;
      =     L      1.2;
      BLD   103;
      AN    M   6260.0;
      AN    M   6280.0;
      AN    M    505.0;
      AN    M    505.1;
      AN    M    505.2;
      A     M    500.2;
      =     L      1.3;
      BLD   103;
      A(    ;
      O     I      0.1;
      O     M   4300.7;
      )     ;
      =     L      1.5;
      BLD   103;
      A     M      0.5;
      =     L      1.6;
      BLD   103;
      CALL #OUT_TRV_CUSHION_B (
           Enable_Aux               := L      0.0,
           Adv_Amount               := 1,
           Ret_Amount               := 1,
           LS_Adv1                  := L      0.1,
           LS_Ret1                  := L      0.2,
           SOL_Adv                  := L      1.1,
           SOL_Ret                  := L      1.2,
           M_Ready                  := L      1.3,
           T_CHK1                   := T#6S,
           T_CHK2                   := T#6S,
           PB_Error_Rst             := L      1.5,
           M_FLICK                  := L      1.6,
           M_Adv_Err                := M    560.4,
           M_Ret_Err                := M    560.5,
           Visu_Adv                 := DB51.DBW   28,
           Visu_Ret                 := DB51.DBW   30);
      NOP   0;
NETWORK
TITLE =

      A     M      3.3;
      =     L      0.0;
      BLD   103;
      A     I     45.1;
      =     L      0.1;
      BLD   103;
      A     I     45.2;
      =     L      0.2;
      BLD   103;
      A     I     45.3;
      =     L      0.4;
      BLD   103;
      A     Q     52.6;
      =     L      1.1;
      BLD   103;
      A     Q     52.7;
      =     L      1.2;
      BLD   103;
      AN    M   6260.0;
      AN    M   6280.0;
      AN    M    505.0;
      AN    M    505.1;
      AN    M    505.2;
      A     M    500.2;
      =     L      1.3;
      BLD   103;
      A(    ;
      O     I      0.1;
      O     M   4300.7;
      )     ;
      =     L      1.5;
      BLD   103;
      A     M      0.5;
      =     L      1.6;
      BLD   103;
      CALL #OUT_TRV_GUIDE (
           Enable_Aux               := L      0.0,
           Adv_Amount               := 1,
           Ret_Amount               := 2,
           LS_Adv1                  := L      0.1,
           LS_Ret1                  := L      0.2,
           LS_Ret2                  := L      0.4,
           SOL_Adv                  := L      1.1,
           SOL_Ret                  := L      1.2,
           M_Ready                  := L      1.3,
           T_CHK1                   := T#8S,
           T_CHK2                   := T#8S,
           PB_Error_Rst             := L      1.5,
           M_FLICK                  := L      1.6,
           M_Adv_Err                := M    560.6,
           M_Ret_Err                := M    560.7,
           Visu_Adv                 := DB51.DBW   32,
           Visu_Ret                 := DB51.DBW   34);
      NOP   0;
NETWORK
TITLE =
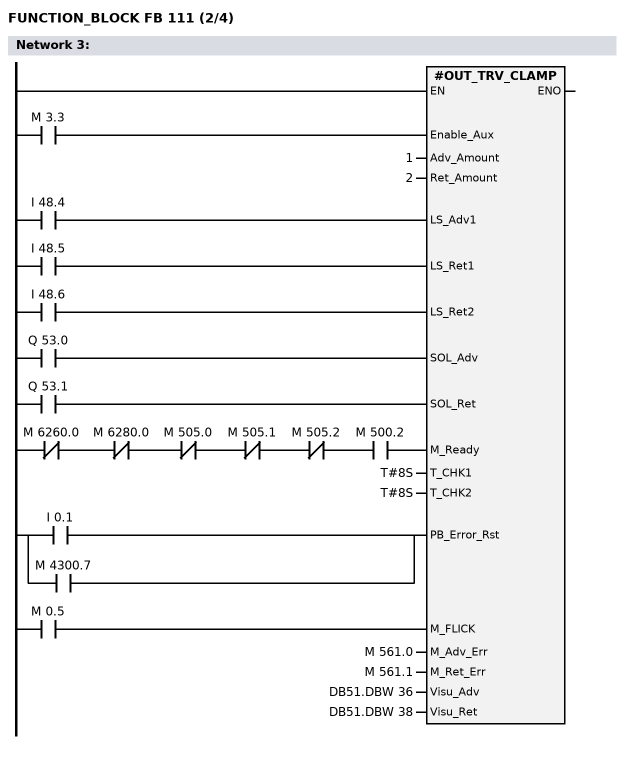

      A     M      3.3;
      =     L      0.0;
      BLD   103;
      A     I     48.4;
      =     L      0.1;
      BLD   103;
      A     I     48.5;
      =     L      0.2;
      BLD   103;
      A     I     48.6;
      =     L      0.4;
      BLD   103;
      A     Q     53.0;
      =     L      1.1;
      BLD   103;
      A     Q     53.1;
      =     L      1.2;
      BLD   103;
      AN    M   6260.0;
      AN    M   6280.0;
      AN    M    505.0;
      AN    M    505.1;
      AN    M    505.2;
      A     M    500.2;
      =     L      1.3;
      BLD   103;
      A(    ;
      O     I      0.1;
      O     M   4300.7;
      )     ;
      =     L      1.5;
      BLD   103;
      A     M      0.5;
      =     L      1.6;
      BLD   103;
      CALL #OUT_TRV_CLAMP (
           Enable_Aux               := L      0.0,
           Adv_Amount               := 1,
           Ret_Amount               := 2,
           LS_Adv1                  := L      0.1,
           LS_Ret1                  := L      0.2,
           LS_Ret2                  := L      0.4,
           SOL_Adv                  := L      1.1,
           SOL_Ret                  := L      1.2,
           M_Ready                  := L      1.3,
           T_CHK1                   := T#8S,
           T_CHK2                   := T#8S,
           PB_Error_Rst             := L      1.5,
           M_FLICK                  := L      1.6,
           M_Adv_Err                := M    561.0,
           M_Ret_Err                := M    561.1,
           Visu_Adv                 := DB51.DBW   36,
           Visu_Ret                 := DB51.DBW   38);
      NOP   0;
NETWORK
TITLE =
